// TwinCAT 3 PLC project Fraktal_Modules
// Title: Fraktal_Modules
// Company: fraktal-automation
// Author: fraktal-automation
// ProjectVersion: 0.11.0.3
// Description: Reusable Fraktal module library: cylinder CMs, clamp EM, simulation models, and configured device presets. Reason bands 10100s/11000s per Core 8.8.
// ProgramVersion: 3.1.4026.24
// libraries:
//   Fraktal_Core, 0.25.0.0 (fraktal-automation)
//   Tc2_MC2, * (Beckhoff Automation GmbH)
//   Tc2_Standard, * (Beckhoff Automation GmbH)
//   Tc2_System, * (Beckhoff Automation GmbH)
//   Tc2_Utilities, * (Beckhoff Automation GmbH)
//   Tc3_Module, * (Beckhoff Automation GmbH)
// project tree:
//   DUTs/ E_ConfigurableCylinderCommand.TcDUT (not stored), E_ClampCommand.TcDUT (not stored), E_CylinderCommand.TcDUT (not stored), E_CylinderPosition.TcDUT (not stored), E_PowerGroupCommand.TcDUT (not stored), ST_TwoHandHal.TcDUT (not stored), ST_TwoHandParCfg.TcDUT (not stored), ST_TwoHandParCmd.TcDUT (not stored), ST_TwoHandOutCmd.TcDUT (not stored), ST_TwoHandOutImm.TcDUT, ST_PowerGroupHal.TcDUT (not stored), ST_PowerGroupParCfg.TcDUT (not stored), ST_PowerGroupParCmd.TcDUT (not stored), ST_PowerGroupOutCmd.TcDUT (not stored), ST_PowerGroupOutImm.TcDUT, ST_ConfigurableCylinderParCfg.TcDUT (not stored), ST_ConfigurableCylinderParCmd.TcDUT (not stored), ST_ConfigurableCylinderOutCmd.TcDUT (not stored), ST_ConfigurableCylinderOutImm.TcDUT, ST_ConfigurableCylinderHal.TcDUT (not stored), ST_ClampParCfg.TcDUT (not stored), ST_ClampParCmd.TcDUT (not stored), ST_ClampOutCmd.TcDUT (not stored), ST_ClampOutImm.TcDUT, ST_CylinderHal.TcDUT (not stored), E_AxisCommand.TcDUT, ST_AxisParCfg.TcDUT, ST_AxisStationCfg.TcDUT, E_RobotOpMode.TcDUT, E_RobotJogMode.TcDUT, E_RobotCommand.TcDUT, E_RobotSimFault.TcDUT, ST_RobotParCfg.TcDUT, ST_RobotParCmd.TcDUT, ST_RobotOutCmd.TcDUT, ST_RobotOutImm.TcDUT, ST_StaubliConnParCfg.TcDUT, ST_RobotPose.TcDUT, E_HelpRole.TcDUT, E_MoveClass.TcDUT, ST_ApproachStep.TcDUT, ST_Corridor.TcDUT, ST_HelpAffinity.TcDUT, ST_NestHelpAffinity.TcDUT, ST_RouteGraph.TcDUT, ST_RobotGeometry.TcDUT, ST_RobotPoint.TcDUT, ST_RobotPointList.TcDUT, ST_AxisParCmd.TcDUT, ST_AxisOutCmd.TcDUT, ST_AxisOutImm.TcDUT, E_SeparatorCommand.TcDUT, E_SeparatorMode.TcDUT, ST_SeparatorHal.TcDUT, ST_SeparatorParCfg.TcDUT, ST_SeparatorParCmd.TcDUT, ST_SeparatorOutCmd.TcDUT, ST_SeparatorOutImm.TcDUT, ST_CylinderParCfg.TcDUT (not stored), ST_CylinderParCmd.TcDUT (not stored), ST_CylinderOutCmd.TcDUT (not stored), ST_CylinderOutImm.TcDUT, ST_CylinderIoIdentity.TcDUT (not stored), ST_DigitalInputHal.TcDUT (not stored), ST_DigitalInputParCfg.TcDUT, ST_DigitalInputParCmd.TcDUT, ST_DigitalInputOutCmd.TcDUT, ST_DigitalInputOutImm.TcDUT, ST_AirPressureHal.TcDUT (not stored), ST_AirPressureStationCfg.TcDUT, ST_AirPressureParCfg.TcDUT, ST_AirPressureParCmd.TcDUT, ST_AirPressureOutCmd.TcDUT, ST_AirPressureOutImm.TcDUT
//   Interfaces/ I_RobotConnector.TcIO
//   / FB_StaubliVal3Connector.TcPOU, FB_RobotRoutePlanner.TcPOU, FB_RobotCM.TcPOU, FB_SimRobotConnector.TcPOU, FB_AxisCM.TcPOU, FB_SeparatorCM.TcPOU, FB_ConfigurableCylinderCM.TcPOU, FB_ConfigurableCylinderSim.TcPOU, FB_ClampEM.TcPOU, FB_CylinderCM.TcPOU, FB_DigitalInputCM.TcPOU, FB_AirPressureMonitorCM.TcPOU, FB_CylinderSim.TcPOU, FB_Iv3VisionCM.TcPOU (not stored), FB_Matrix220CM.TcPOU (not stored), FB_PowerGroupCM.TcPOU, FB_TwoHandStartCM.TcPOU
//   Params/ PL_RobotPlanner.TcGVL, PL_ModuleReasons.TcGVL
// real-time tasks:
//   TASK PlcTask: cycle T#10ms, priority 20, ADS port 350

// ---- DUTs/ST_TwoHandOutImm.TcDUT
TYPE ST_TwoHandOutImm :
STRUCT
    LeftPressed     : BOOL;
    RightPressed    : BOOL;
    SafeActive      : BOOL;
    Armed           : BOOL;
    StartPulse      : BOOL;
    FieldbusHealthy : BOOL;
END_STRUCT
END_TYPE

// ---- DUTs/ST_PowerGroupOutImm.TcDUT
TYPE ST_PowerGroupOutImm :
STRUCT
    Status     : ST_PowerGroupStatus;
END_STRUCT
END_TYPE

// ---- DUTs/ST_ConfigurableCylinderOutImm.TcDUT
TYPE ST_ConfigurableCylinderOutImm :
STRUCT
    Position   : E_CylinderPosition;
    AtHome     : BOOL;
    AtWork     : BOOL;
END_STRUCT
END_TYPE

// ---- DUTs/ST_ClampOutImm.TcDUT
TYPE ST_ClampOutImm :
STRUCT
    Clamped    : BOOL;
    Unclamped  : BOOL;
END_STRUCT
END_TYPE

// ---- DUTs/E_AxisCommand.TcDUT
{attribute 'qualified_only'}
// Annex G motion CM. NONE is the unset value: dispatch rejects it (S5.6).
TYPE E_AxisCommand : (
    NONE    := 0,
    HOME    := 1,
    MOVE_TO := 2,
    // HELD commands (§7.6.1). Two entries rather than one plus a direction, so
    // the generic HMI renders two hold-buttons with no axis-specific code.
    // They never reach _M_Dispatch: a jog is not an Execute/Done command, and
    // PLCopen models it with level inputs for the same reason.
    JOG_POS := 3,
    JOG_NEG := 4
) DINT;
END_TYPE

// ---- DUTs/ST_AxisParCfg.TcDUT
// Core S3.8: SchemaVersion FIRST. Soft limits and dynamics are recipe/config,
// never sequence literals (S10.3) - scaling and hard limits stay in the axis
// configuration where the drive integrator owns them.
TYPE ST_AxisParCfg :
STRUCT
    SchemaVersion : UINT := 1;
    SoftMin       : LREAL := 0.0;
    SoftMax       : LREAL := 100.0;
    Velocity      : LREAL := 50.0;
    Acceleration  : LREAL := 500.0;
    Deceleration  : LREAL := 500.0;
    MoveTimeout   : TIME := T#10S;
    HomeTimeout   : TIME := T#30S;
    // Teach jog (§7.6.1). JogVelocity is DEFENCE IN DEPTH, not the protection:
    // the safety-rated reduced speed is the drive's own SLS or the cell's safe
    // speed monitor, because a scan overrun or a download must not be able to
    // remove the limit that keeps a person safe (§9).
    JogVelocity     : LREAL := 5.0;
    JogAcceleration : LREAL := 100.0;
    // How long a held request may go unheard before the axis stops. This is the
    // backstop for a stalled transport, NOT the normal stop: releasing the
    // control sends Dir=0 and stops immediately (O10).
    JogTimeout      : TIME := T#200MS;
END_STRUCT
END_TYPE

// ---- DUTs/ST_AxisStationCfg.TcDUT
// Core §3.8a/§3.8b - deployment data for one axis: what this MACHINE is, as
// opposed to what the current product needs. A taught position belongs here and
// not in ParCfg, because I_RecipeProvider loads and never stores: the next
// changeover would overwrite a number an operator spent time teaching.
//
// SchemaVersion is FIRST and is mandatory (§3.8b). Version 0 means never
// written - a first boot has lost nothing. Any OTHER unrecognized version means
// a real image was rejected, which is annunciated, because the difference
// between an empty machine and one that has just lost its commissioning is
// exactly what an operator needs told.
TYPE ST_AxisStationCfg :
STRUCT
    SchemaVersion  : UINT;      // 0 = never written; 2 = this layout
    TaughtPosition : LREAL;     // captured from the live ActPos (§3.8c)
    // v2. Does THIS INSTALLATION have a safety-rated enabling device for manual
    // motion? A deployment fact, not a preference, which is why it is station
    // configuration (§3.8a) rather than a recipe value or a compiled-in
    // assumption in the reusable type.
    //
    // TRUE - the default, and what every restore that predates this member and
    // every rejected image falls back to - keeps the §G.4a rule: no enabling
    // device permitting, no jog. FALSE says this installation has none, and a
    // station shall declare that only when it is true AND the consequence has
    // been assessed: a bench with a low-force motor on a desk is the case it
    // exists for, a cell with a person inside it is not. A station declaring
    // FALSE should declare a §7.5 engineering gate with it, so the machine
    // annunciates the departure instead of hiding it in a value nobody reads.
    JogRequiresEnable : BOOL;
END_STRUCT
END_TYPE

// ---- DUTs/E_RobotOpMode.TcDUT
// Annex I I.4a(a) - the robot CONTROLLER's operating mode, which bounds what
// motion is physically allowed. The PLC REQUESTS a mode and publishes separately
// what the controller REPORTS it actually is: a request that was not granted must
// stay visibly ungranted, never overwritten by optimism. UNKNOWN = 0 so an
// uninitialised value is never mistaken for a permissive mode.
{attribute 'qualified_only'}
TYPE E_RobotOpMode :
(
    UNKNOWN        := 0,
    AUTO_REMOTE    := 1,
    MANUAL_REDUCED := 2,
    MANUAL_HIGH    := 3
) DINT;
END_TYPE

// ---- DUTs/E_RobotJogMode.TcDUT
// Annex I I.3 - jog frame for manual motion. Named E_RobotJogMode, not
// E_JogMode: the short name collides with a Beckhoff motion-library type and the
// ambiguity surfaces only in a consumer that references both. Manual only, release-gated (S7.6).
{attribute 'qualified_only'}
TYPE E_RobotJogMode :
(
    JOINT     := 0,
    CARTESIAN := 1,
    TOOL      := 2
) DINT;
END_TYPE

// ---- DUTs/E_RobotCommand.TcDUT
// Annex I I.4 - the robot CM's command vocabulary. A point, a taught path, a
// generated route or a pallet nest is ONE command that runs to completion, so the
// robot looks identical to any other CM (S6.1). IDs are the only addressing.
{attribute 'qualified_only'}
TYPE E_RobotCommand :
(
    NONE           := 0,
    POWER_ON       := 1,
    POWER_OFF      := 2,
    HOME           := 3,
    MOVE_TO        := 4,   // one taught point, by ID
    RUN_PATH       := 5,   // a stored list, by ID and optional sub-range
    RUN_PALLET     := 6,   // one nest of a generated pallet grid
    MOVE_TEMPLATE  := 7,   // route generated by the help/nest graph (I.9)
    MOVE_FROM_AREA := 8,   // start resolved live from the current area (I.11)
    SET_TOOL       := 9,
    SET_FRAME      := 10,
    RECONNECT      := 11   // §3.15.4 deliberate reconnect; never resumes a command
) DINT;
END_TYPE

// ---- DUTs/E_RobotSimFault.TcDUT
// Annex I I.5c - the failures the simulation connector can be told to inject.
// Bounded and enumerated (O10): the reasons of I.2 are exactly what cannot be
// proven against a real arm without deliberately breaking a cell, so the sim
// must be able to produce them on demand - but only the ones some test or
// commissioning rehearsal actually needs, never a knob per reason.
{attribute 'qualified_only'}
TYPE E_RobotSimFault :
(
    NONE            := 0,
    POINT_UNREACHABLE := 1,   // the next motion command is refused before it starts
    NO_ROUTE          := 2,   // the next template move finds no path (I.9)
    LINK_LOSS         := 3,   // the heartbeat fails; the base drops and re-backs off
    PROTECTIVE_STOP   := 4,   // the crash device trips, in motion or at rest
    NOT_RESUMABLE     := 5    // a held move cannot resume - the arm left the path (I.4b)
) DINT;
END_TYPE

// ---- DUTs/ST_RobotParCfg.TcDUT
// Recipe-class configuration (S3.8), versioned.
TYPE ST_RobotParCfg :
STRUCT
    SchemaVersion : UINT := 1;
    MoveTimeout   : TIME := T#60S;   // per-command guard; the Unit step's ExpectedTime (S6.5) remains the outer one
    HomeTimeout   : TIME := T#120S;
    SpeedScaleMin : REAL := 1.0;     // band a recipe SpeedScale is validated against (I.4a(b))
    SpeedScaleMax : REAL := 100.0;
    // Ceiling per controller operating mode; the CM applies MIN(ceiling, ParCmd.SpeedScale).
    // UNKNOWN = 0 so an unreported mode yields the safest ceiling, not the fastest.
    // Indexed by E_RobotOpMode's ordinals - UNKNOWN, AUTO_REMOTE,
    // MANUAL_REDUCED, MANUAL_HIGH. UNKNOWN is 0.0 on purpose: a mode the
    // controller has not reported never earns a speed allowance.
    SpeedCeiling  : ARRAY[0..3] OF REAL := [0.0, 100.0, 25.0, 100.0];
END_STRUCT
END_TYPE

// ---- DUTs/ST_RobotParCmd.TcDUT
// Latched by the base on the Execute rising edge (S6.1). No Offset field yet:
// the runtime-correction exception of I.8a is deferred with the connector support
// for it - declaring a field no consumer reads would be dead surface, and an
// unvalidated offset would be worse (S14).
TYPE ST_RobotParCmd :
STRUCT
    TargetId   : DWORD := 0;   // point / list / pallet / tool / frame - or the TO position
    FromId     : DWORD := 0;   // FROM position (MOVE_TEMPLATE only)
    Nest       : DINT := 0;    // nest index (RUN_PALLET only)
    StartIdx   : DINT := -1;   // sub-path bounds (RUN_PATH; -1,-1 = whole list)
    EndIdx     : DINT := -1;
    SpeedScale : REAL := 100.0;   // process speed for THIS command, % of taught (I.4a(b))
    AcknowledgeController : BOOL; // RECONNECT also clears the robot's own fault
END_STRUCT
END_TYPE

// ---- DUTs/ST_RobotOutCmd.TcDUT
// Valid on Done (S3.10).
TYPE ST_RobotOutCmd :
STRUCT
    ReachedId : DWORD;   // position actually reached
END_STRUCT
END_TYPE

// ---- DUTs/ST_RobotOutImm.TcDUT
// Cyclic live status mirrored from the connector, plus the first-out diagnostic.
TYPE ST_RobotOutImm :
STRUCT
    Linked         : BOOL;
    Referenced     : BOOL;
    MotionBusy     : BOOL;           // the ARM is moving - not the command handshake
    ActualMode     : E_RobotOpMode;  // what the controller REPORTS (I.4a(a))
    CurrentArea    : DWORD;          // 0 = none/undefined (I.11)
    ProtectiveStop : BOOL;           // process protection, NOT S9 safety (I.4a(c))
    Resumable      : BOOL;           // resume still valid on the retained path (I.4b)
    SpeedScale     : REAL;           // scale actually in force
END_STRUCT
END_TYPE

// ---- DUTs/ST_StaubliConnParCfg.TcDUT
// Deployment configuration for the VAL3 connector (S3.8a station config).
TYPE ST_StaubliConnParCfg :
STRUCT
    SchemaVersion : UINT := 1;
    Host          : STRING(80);
    Port          : UINT := 11000;      // VAL3 fraktal_server command socket
    Terminator    : STRING(2) := '$R';  // ASCII 13, as the Staubli sioLink default
    RespTimeout   : TIME := T#2S;       // per-request; motion completion is polled, not awaited
    StatusPeriod  : TIME := T#100MS;    // idle status poll interval
END_STRUCT
END_TYPE

// ---- DUTs/ST_RobotPose.TcDUT
// Annex I I.3 - one pose type for live readback, taught geometry and runtime
// corrections. The connector owns the Euler convention and the units it speaks
// to the controller in; per-model facts like that are data it reads, never
// branches in application code.
TYPE ST_RobotPose :
STRUCT
    X  : LREAL;   // mm
    Y  : LREAL;
    Z  : LREAL;
    RX : LREAL;   // deg
    RY : LREAL;
    RZ : LREAL;
END_STRUCT
END_TYPE

// ---- DUTs/E_HelpRole.TcDUT
// Annex I I.10 - which direction of travel a help corridor is legal for.
// EITHER is 0 so a zero-initialized corridor is bidirectional: a nest is
// exit-able the way it was entered unless its geometry is physically one-way.
{attribute 'qualified_only'}
TYPE E_HelpRole :
(
    EITHER   := 0,
    APPROACH := 1,
    DEPART   := 2
) DINT;
END_TYPE

// ---- DUTs/E_MoveClass.TcDUT
// Annex I I.10.2 - how a generated step is flown. The class selects the motion
// mode AND which configured velocity applies, so speed stays configuration
// (I.4a(b)) and never becomes a literal in the route graph.
{attribute 'qualified_only'}
TYPE E_MoveClass :
(
    SLOW_LINEAR := 0,
    FAST_PTP    := 1,
    SLOW_JOINTS := 2
) DINT;
END_TYPE

// ---- DUTs/ST_ApproachStep.TcDUT
// Annex I I.10.2 - one offset from the nest pose, in the nest's own frame.
TYPE ST_ApproachStep :
STRUCT
    D         : ST_RobotPose;   // offset applied to the nest pose
    MoveClass : E_MoveClass;
END_STRUCT
END_TYPE

// ---- DUTs/ST_Corridor.TcDUT
// Annex I I.10.2 - how a nest is entered from, or left toward, one serving
// help. Steps are stored nest-ward -> help-ward: a DEPART corridor emits them
// in that order, an APPROACH corridor emits them reversed and then the nest.
// StepCount = 0 with ListId <> 0 names a taught list instead, for geometry a
// few axis offsets cannot express.
TYPE ST_Corridor :
STRUCT
    Steps     : ARRAY[1..PL_RobotPlanner.MAX_APPROACH_STEPS] OF ST_ApproachStep;
    StepCount : INT;
    ListId    : DWORD;
END_STRUCT
END_TYPE

// ---- DUTs/ST_HelpAffinity.TcDUT
// Annex I I.10 - one help point serving a nest, with the direction it is legal
// for and the transit region it connects to. Region is needed only where a nest
// has two corridors for the SAME direction; most nests need only the role.
TYPE ST_HelpAffinity :
STRUCT
    HelpId   : INT;          // index into the help arrays; 0 = unused entry
    Role     : E_HelpRole;
    RegionId : DWORD;        // 0 = any
    Approach : ST_Corridor;  // how the nest is ENTERED from this help
    Depart   : ST_Corridor;  // how it is LEFT toward this help - not the approach reversed
END_STRUCT
END_TYPE

// ---- DUTs/ST_NestHelpAffinity.TcDUT
// Annex I I.10 - the help points serving one nest. Count = 1 is the trivial
// single-help case; multi-help is the general one.
TYPE ST_NestHelpAffinity :
STRUCT
    Helps : ARRAY[1..PL_RobotPlanner.MAX_HELPS_PER_NEST] OF ST_HelpAffinity;
    Count : INT;
END_STRUCT
END_TYPE

// ---- DUTs/ST_RouteGraph.TcDUT
// Annex I I.9 / Core S10.7 - the declarative routing model. The application
// supplies configuration, not traversal code: one generic planner resolves it
// for every station.
TYPE ST_RouteGraph :
STRUCT
    // help <-> help adjacency: which transits are allowed
    HelpAdj    : ARRAY[1..PL_RobotPlanner.MAX_HELPS, 1..PL_RobotPlanner.MAX_HELPS] OF BOOL;
    // the transit region each help belongs to; used only to break ties between
    // same-direction corridors (I.10)
    HelpRegion : ARRAY[1..PL_RobotPlanner.MAX_HELPS] OF DWORD;
    // per gripper, per nest: one OR MORE serving help points (I.10, I.12)
    NestHelp   : ARRAY[1..PL_RobotPlanner.MAX_GRIPPERS, 1..PL_RobotPlanner.MAX_NESTS] OF ST_NestHelpAffinity;
    // optional taught nest -> nest list, bypassing the help routing entirely
    DirectNest : ARRAY[1..PL_RobotPlanner.MAX_NESTS, 1..PL_RobotPlanner.MAX_NESTS] OF DWORD;
END_STRUCT
END_TYPE

// ---- DUTs/ST_RobotGeometry.TcDUT
// Annex I I.1 - taught geometry held as Fraktal configuration and pushed to the
// controller by the connector, so it lives inside changeover (S3.8), parameter
// sets (S3.8b), access control (S7.7) and audit (S8.3) rather than only inside a
// vendor engineering tool. Editable through bounded collection capabilities
// (S3.10.2a) with pose cells filled by teach capture (S3.8c).
TYPE ST_RobotGeometry :
STRUCT
    HelpPose : ARRAY[1..PL_RobotPlanner.MAX_HELPS] OF ST_RobotPose;
    NestPose : ARRAY[1..PL_RobotPlanner.MAX_GRIPPERS, 1..PL_RobotPlanner.MAX_NESTS] OF ST_RobotPose;
END_STRUCT
END_TYPE

// ---- DUTs/ST_RobotPoint.TcDUT
// Annex I I.8 - one element of a generated or taught route. A point either
// names a pose to move to, or (ListId <> 0) a taught list for the executor to
// run at that place in the sequence.
TYPE ST_RobotPoint :
STRUCT
    Target    : ST_RobotPose;
    MoveClass : E_MoveClass;
    ListId    : DWORD;    // 0 = move to Target; otherwise run this taught list
END_STRUCT
END_TYPE

// ---- DUTs/ST_RobotPointList.TcDUT
// Annex I I.8 - a bounded generated or taught route.
TYPE ST_RobotPointList :
STRUCT
    Points : ARRAY[1..PL_RobotPlanner.MAX_ROUTE_POINTS] OF ST_RobotPoint;
    Count  : INT;
END_STRUCT
END_TYPE

// ---- DUTs/ST_AxisParCmd.TcDUT
// Latched by the base on the Execute rising edge (S6.1).
TYPE ST_AxisParCmd :
STRUCT
    Target : LREAL;   // absolute target for MOVE_TO, in axis units
END_STRUCT
END_TYPE

// ---- DUTs/ST_AxisOutCmd.TcDUT
// Valid on Done (S3.12).
TYPE ST_AxisOutCmd :
STRUCT
    InPosition : BOOL;
    Homed      : BOOL;
END_STRUCT
END_TYPE

// ---- DUTs/ST_AxisOutImm.TcDUT
// Cyclic live status plus the first-out diagnostic (S3.12, S6.9).
TYPE ST_AxisOutImm :
STRUCT
    ActPos       : LREAL;
    ActVelocity  : LREAL;
    Homed        : BOOL;
    DriveEnabled : BOOL;
    // The stored taught position (S3.8b PERSISTENT), published beside the live
    // ActPos so an operator can compare what is stored with where the axis is
    // before capturing over it (S3.8c(b)).
    TaughtPosition : LREAL;
    Jogging      : BOOL;   // a held jog is driving the axis right now (§7.6.1)
    // Why the last jog stopped: 0 = released normally, otherwise the §8.8 reason.
    // Published status, deliberately NOT an alarm - a jog that stops because the
    // operator let go is the designed behaviour, and filing it as a fault would
    // fill the record with events that were never faults (§6.1).
    JogStopReason : DINT;
END_STRUCT
END_TYPE

// ---- DUTs/E_SeparatorCommand.TcDUT
{attribute 'qualified_only'}
// Annex A separator/stopper. NONE is the unset value: dispatch rejects it (S5.6).
TYPE E_SeparatorCommand : (
    NONE       := 0,
    SEPARATE   := 1,    // release exactly one carrier
    OPEN_CLOSE := 2     // hold the stopper open or closed per ParCmd.OpenStopper
) DINT;
END_TYPE

// ---- DUTs/E_SeparatorMode.TcDUT
{attribute 'qualified_only'}
// Separation behaviour variants (Annex A). SEPARATOR checks the carrier at AND
// after the device; STOPPER checks only at it.
TYPE E_SeparatorMode : (
    SEPARATOR  := 0,
    STOPPER    := 1,
    ASISTOPPER := 2,
    LEADFRAME  := 3
) DINT;
END_TYPE

// ---- DUTs/ST_SeparatorHal.TcDUT
// HAL view (S10.3). The driver owns invert/debounce and the raw %I/%Q symbols;
// the module only ever touches these clean signals, so simulation and hardware
// are the same code (S2.6).
TYPE ST_SeparatorHal :
STRUCT
    CarrierAt    : BOOL;   // input  - carrier present at the separator
    CarrierAfter : BOOL;   // input  - carrier present just past the separator
    OpenedFb     : BOOL;   // input  - separator-opened feedback (optional)
    ValveOpen    : BOOL;   // output - drives the open solenoid
END_STRUCT
END_TYPE

// ---- DUTs/ST_SeparatorParCfg.TcDUT
// Core S3.8: SchemaVersion FIRST, initialized to the expected version.
TYPE ST_SeparatorParCfg :
STRUCT
    SchemaVersion : UINT := 1;
    Mode          : E_SeparatorMode := E_SeparatorMode.SEPARATOR;
    CheckAfter    : BOOL := TRUE;    // require the carrier-after arrival/clear checks
    UsesOpenFb    : BOOL := FALSE;   // require the open feedback on OPEN_CLOSE
    MaxOpenTime   : TIME := T#3S;    // CarrierAt must clear within this after opening
    SOnMaxTime    : TIME := T#3S;    // CarrierAfter must arrive/clear within this
    CloseDelay    : TIME := T#0S;
    Timeout       : TIME := T#10S;   // overall command timeout
END_STRUCT
END_TYPE

// ---- DUTs/ST_SeparatorParCmd.TcDUT
// Latched by the base on the Execute rising edge (S6.1).
TYPE ST_SeparatorParCmd :
STRUCT
    OpenStopper : BOOL;   // OPEN_CLOSE: TRUE = open, FALSE = close
END_STRUCT
END_TYPE

// ---- DUTs/ST_SeparatorOutCmd.TcDUT
// Valid on Done (S3.12).
TYPE ST_SeparatorOutCmd :
STRUCT
    SeparateOk    : BOOL;
    SeparatorOpen : BOOL;
END_STRUCT
END_TYPE

// ---- DUTs/ST_SeparatorOutImm.TcDUT
// Cyclic live status plus the first-out diagnostic (S3.12, S6.9).
TYPE ST_SeparatorOutImm :
STRUCT
    CarrierAt    : BOOL;
    CarrierAfter : BOOL;
    OpenedFb     : BOOL;
    ValveOpen    : BOOL;
END_STRUCT
END_TYPE

// ---- DUTs/ST_CylinderOutImm.TcDUT
TYPE ST_CylinderOutImm :
STRUCT
    Extended   : BOOL;
    Retracted  : BOOL;
    ExtendedSensorTag : STRING(80);
    RetractedSensorTag: STRING(80);
    ExtendOutputTag   : STRING(80);
    RetractOutputTag  : STRING(80);
END_STRUCT
END_TYPE

// ---- DUTs/ST_DigitalInputParCfg.TcDUT
TYPE ST_DigitalInputParCfg :
STRUCT
    SchemaVersion : UINT := 1; // §3.8: first member even when the passive type has no behavior parameter
END_STRUCT
END_TYPE

// ---- DUTs/ST_DigitalInputParCmd.TcDUT
TYPE ST_DigitalInputParCmd :
STRUCT
    Reserved : BOOL; // passive monitor: physical four-structure contract, no command payload
END_STRUCT
END_TYPE

// ---- DUTs/ST_DigitalInputOutCmd.TcDUT
TYPE ST_DigitalInputOutCmd :
STRUCT
    Reserved : BOOL; // passive monitor: no command result
END_STRUCT
END_TYPE

// ---- DUTs/ST_DigitalInputOutImm.TcDUT
TYPE ST_DigitalInputOutImm :
STRUCT
    Value : BOOL;
    Quality : BOOL;
    IoTag : STRING(80);
END_STRUCT
END_TYPE

// ---- DUTs/ST_AirPressureStationCfg.TcDUT
// Core §3.8a/§3.8b — deployment data for this monitor. The qualification time
// depends on the physical switches and the air system they sit in, not on the
// product being made, so it is station configuration and NOT part of any model
// recipe: it must not change at changeover, and it must survive a restart.
// SchemaVersion stays first (§3.8b) so a retained image from another layout is
// rejected and re-initialized instead of read by field position.
TYPE ST_AirPressureStationCfg :
STRUCT
    SchemaVersion : UINT := 1;
    ConflictTime  : TIME := T#500MS; // qualify contradictory mechanical switches
END_STRUCT
END_TYPE

// ---- DUTs/ST_AirPressureParCfg.TcDUT
// v2 moved ConflictTime to ST_AirPressureStationCfg: it varies per
// deployment, not per model, and §3.8a places such a value in station
// configuration. This monitor has no model data of its own, so what remains
// is the versioned shell the §3.12 contract asks every module to carry.
TYPE ST_AirPressureParCfg :
STRUCT
    SchemaVersion : UINT := 2;       // §3.8: MUST remain first
END_STRUCT
END_TYPE

// ---- DUTs/ST_AirPressureParCmd.TcDUT
TYPE ST_AirPressureParCmd :
STRUCT
    Reserved : BOOL; // passive monitor: physical four-structure contract, no command payload
END_STRUCT
END_TYPE

// ---- DUTs/ST_AirPressureOutCmd.TcDUT
TYPE ST_AirPressureOutCmd :
STRUCT
    Reserved : BOOL; // passive monitor: no command result
END_STRUCT
END_TYPE

// ---- DUTs/ST_AirPressureOutImm.TcDUT
TYPE ST_AirPressureOutImm :
STRUCT
    LowPressure : BOOL;
    OperatingPressure : BOOL;
    PressureOk : BOOL;
    Contradictory : BOOL;
    Quality : BOOL;
    LowSensorTag : STRING(80);
    OperatingSensorTag : STRING(80);
END_STRUCT
END_TYPE

// ---- Params/PL_RobotPlanner.TcGVL
{attribute 'qualified_only'}
// Annex I - bounds for the declarative routing model. Every structure the
// planner touches is statically sized (Core S1.1 O10): a route that would
// exceed MAX_ROUTE_POINTS is refused, never allocated.
VAR_GLOBAL CONSTANT
    MAX_HELPS           : INT := 8;    // transit / wait positions
    MAX_NESTS           : INT := 16;   // work positions, per gripper
    MAX_GRIPPERS        : INT := 4;    // nests are per-gripper (I.12); 1 is the trivial case
    MAX_HELPS_PER_NEST  : INT := 4;    // serving corridors on one nest (I.10)
    MAX_APPROACH_STEPS  : INT := 4;    // offset steps in one corridor (I.10.2)
    MAX_ROUTE_POINTS    : INT := 32;   // generated route length
END_VAR

// ---- Params/PL_ModuleReasons.TcGVL
{attribute 'qualified_only'}
// Core §8.8 band constants (band-extensibility rule): cylinder CM 10100-10199,
// clamp EM 11000-11999 — registered in the Core §8.8 registry.
VAR_GLOBAL CONSTANT
    CYL_NOT_EXTENDED    : DINT := 10101;
    CYL_NOT_RETRACTED   : DINT := 10102;
    CYL_BOTH_SENSORS    : DINT := 10103;
    CLAMP_NOT_CONFIRMED : DINT := 11001;
    // basic cylinder 10110-10119
    CYL_HOME_NOT_REACHED : DINT := 10111;   // timeout moving to home
    CYL_WORK_NOT_REACHED : DINT := 10112;   // timeout moving to work
    CYL_POS_IMPLAUSIBLE  : DINT := 10113;   // home AND work sensor confirmed at once (implausible)
    CYL_SENSOR_LOST      : DINT := 10114;   // confirmed position sensor dropped while holding
    CYL_DISCREPANCY      : DINT := 10116;   // redundant sensors for one position disagree > DiscrepancyTime
    CYL_CFG_INVALID      : DINT := 10115;   // TravelTime >= MoveTimeout, or no sensor+no travel
    // axis CM 10201-10206 (Annex G)
    AXIS_TARGET_OOR      : DINT := 10201;   // target outside soft limits (rejected)
    AXIS_MOVE_TIMEOUT    : DINT := 10202;   // MC move did not complete within the timeout
    AXIS_DRIVE_FAULT     : DINT := 10203;   // MC_* .Error / drive fault
    AXIS_NOT_HOMED       : DINT := 10204;   // MOVE_TO before a valid home
    AXIS_JOG_NOT_ENABLED : DINT := 10205;   // teach jog asked with no enabling device held
    AXIS_JOG_RELEASED    : DINT := 10206;   // the held jog request stopped arriving
    // power-group CM 10500-10599
    POWER_ENABLE_WITHHELD : DINT := 10501;
    POWER_FEEDBACK_TIMEOUT: DINT := 10502;
    // separator/stopper CM 10001-10005 (Annex A)
    SEP_NO_CARRIER_AT       : DINT := 10001;   // carrier never present at the separator
    SEP_CARRIER_NOT_CLEARED : DINT := 10002;   // CarrierAt did not clear after opening
    SEP_CARRIER_NOT_ARRIVED : DINT := 10003;   // CarrierAfter did not arrive in time
    SEP_NOT_OPENED_FB       : DINT := 10004;   // open feedback missing
    SEP_SON_NOT_CLEARED     : DINT := 10005;   // CarrierAfter did not clear after close
    // robot route planner 10301-10315 (Annex I) - only what the planner raises today
    ROBOT_POINT_UNREACHABLE  : DINT := 10301;   // taught point not reachable with the active tool/frame
    ROBOT_MOVE_TIMEOUT       : DINT := 10303;   // motion did not complete within ParCfg timeout
    ROBOT_CONTROLLER_FAULT   : DINT := 10304;   // drive/controller fault reported by the robot itself
    ROBOT_NOT_REFERENCED     : DINT := 10305;   // motion commanded before a valid home/reference
    ROBOT_NO_ROUTE           : DINT := 10308;   // help graph defines no path between the two positions
    ROBOT_NO_HELP_FOR_NEST   : DINT := 10310;   // no help point resolves for a nest given the move endpoints
    ROBOT_MODE_NOT_PERMITTED : DINT := 10311;   // controller mode does not permit this command
    ROBOT_PROTECTIVE_STOP    : DINT := 10313;   // collision/crash device tripped - NOT a S9 safety function
    ROBOT_PARAM_OOR          : DINT := 10314;   // a command parameter is outside its configured band
    ROBOT_RESUME_INVALID     : DINT := 10315;   // resume after hold, but the arm left the retained path
    // air-pressure monitor CM 10600-10699
    AIR_SWITCH_CONFLICT    : DINT := 10601;
END_VAR

// ---- Interfaces/I_RobotConnector.TcIO
// Annex I I.3 - the primitive robot surface, below the robot CM and above the
// protocol. Everything under it (transport, point database, kinematics, path
// planning) is confined to the implementation (Core S3.15).
//
// MOST OF THIS SURFACE IS NOT FRAKTAL'S TO DEFINE. SRCI (Standard Robot Command
// Interface, PROFIBUS/PROFINET International) already standardises the PLC/robot
// command boundary, so the members below are DEFINED BY their SRCI equivalent and
// are not re-described here - re-describing them would create a second authority
// for someone else's contract and guarantee drift (S1.1 O9). The mapping is
// normative and lives in Annex I I.3:
//
//   PowerOn/PowerOff  = EnableRobot        Interrupt/Resume = GroupInterrupt/Continue
//   Home              = referencing        Abort            = GroupStop
//   MoveToPoint       = MoveDirectAbsolute ResetController  = GroupReset
//   RunPath           = sequential moves   RequestMode      = SetOperationMode
//   ActualPosition    = ReadActualPosition SetSpeedScale    = ChangeSpeedOverride
//   ControllerMessage = ReadMessages       SetTool/SetFrame = Read Tool/FrameData
//   SetPayload        = Read/WriteLoadData Jog              = GroupJog
//
// Seven members have NO SRCI equivalent, because they express this annex's own
// model: RunPallet, MoveTemplate, MoveFromArea, CurrentArea, ProtectiveStop,
// Resumable and LastResult. They are what the standard adds over an ordinary
// robot command interface.
//
// Every method returns immediately: FALSE means the request was refused outright
// (unknown id, unreachable, no route, not linked) and LastResult carries the
// first-out reason. Motion progress is observed over scans via Busy, never awaited.
INTERFACE I_RobotConnector EXTENDS I_DeviceConnector

// SRCI EnableRobot (Core). Arm power on.
METHOD PowerOn : BOOL
END_METHOD

// SRCI EnableRobot (Core). Arm power off.
METHOD PowerOff : BOOL
END_METHOD

// SRCI referencing. Drive to the home/reference configuration.
METHOD Home : BOOL
END_METHOD

// SRCI MoveDirectAbsolute/MoveLinearAbsolute, target resolved from the ID.
METHOD MoveToPoint : BOOL
VAR_INPUT
    PointId : DWORD;
END_VAR
END_METHOD

// Sequential SRCI moves over a stored list. (-1,-1) = the whole list.
METHOD RunPath : BOOL
VAR_INPUT
    ListId   : DWORD;
    StartIdx : DINT;
    EndIdx   : DINT;
END_VAR
END_METHOD

// SRCI GroupInterrupt (Core). Stop ON PATH, retaining the resume point - the
// robot half of the S6.1 HELD contract (I.4b). A cylinder honours HELD by
// de-energising; a robot cannot, because resuming a 26-point path by
// re-commanding it would re-run executed points or approach from an untaught pose.
METHOD Interrupt : BOOL
END_METHOD

// SRCI GroupContinue (Core). Continue FROM the retained path point. Callers
// must check Resumable first: resuming onto a path the tool has left is how a
// robot drives through a fixture (I.4b).
METHOD Resume : BOOL
END_METHOD

// SRCI GroupStop (Core). Commands are NOT auto-repeated; resumption is
// deliberate (Annex D / S9.3).
METHOD Abort : BOOL
END_METHOD

// SRCI GroupReset (Core). Acknowledge the robot's OWN messages. Without this a
// controller fault can be detected but never cleared.
METHOD ResetController : BOOL
END_METHOD

// SRCI SetOperationMode (Core). REQUEST only - the controller grants. Compare
// with ActualMode, which reports what it actually is (I.4a(a)).
METHOD RequestMode : BOOL
VAR_INPUT
    Mode : E_RobotOpMode;
END_VAR
END_METHOD

// SRCI ChangeSpeedOverride (Core). Ceiling on path speed, as a percentage of
// taught. The CM applies MIN(mode ceiling, recipe scale) (I.4a(b)).
METHOD SetSpeedScale : BOOL
VAR_INPUT
    Percent : REAL;
END_VAR
END_METHOD

// SRCI ReadToolData (Core) - selection by ID. Geometry stays taught data.
METHOD SetTool : BOOL
VAR_INPUT
    ToolId : DWORD;
END_VAR
END_METHOD

// SRCI ReadFrameData (Core) - selection by ID. The frame may be chained (I.12).
METHOD SetFrame : BOOL
VAR_INPUT
    FrameId : DWORD;
END_VAR
END_METHOD

// SRCI Read/WriteLoadData. The active load case, which changes the moment a part
// is gripped or released; a move computed for the wrong mass degrades accuracy
// and brake margin silently (I.3).
METHOD SetPayload : BOOL
VAR_INPUT
    LoadId : DWORD;
END_VAR
END_METHOD

// SRCI GroupJog (Core). Manual only, release-gated (S7.6), and refused unless
// ActualMode is a manual mode (I.4a(a)).
METHOD Jog : BOOL
VAR_INPUT
    Mode : E_RobotJogMode;
    Axis : INT;
    Dir  : INT;
END_VAR
END_METHOD

// NO SRCI EQUIVALENT. One nest of a generated pallet grid, addressed by pallet
// ID and nest index; the grid itself is generated from taught corners (I.12).
METHOD RunPallet : BOOL
VAR_INPUT
    PalletId : DWORD;
    Nest     : DINT;
END_VAR
END_METHOD

// NO SRCI EQUIVALENT. Route generated by the declarative help/nest graph between
// two KNOWN positions (I.9) - the PLC names from and to, never the waypoints.
METHOD MoveTemplate : BOOL
VAR_INPUT
    FromPosId : DWORD;
    ToPosId   : DWORD;
END_VAR
END_METHOD

// NO SRCI EQUIVALENT. Route planned from WHICHEVER planning area the TCP
// currently occupies, resolved live. The application's primary motion command,
// because it needs no assumption about the start pose; pose recovery after an
// E-stop is its extreme case, not a separate mode (I.11).
METHOD MoveFromArea : BOOL
VAR_INPUT
    ToPosId : DWORD;
END_VAR
END_METHOD

// The ROBOT is executing motion. Deliberately NOT called Busy: the module base
// already publishes Busy for its own command handshake, and the two are different
// questions - "is my command running" versus "is the arm moving".
PROPERTY MotionBusy : BOOL
GET
END_GET
END_PROPERTY

// A valid home/reference exists. MOVE/RUN before this is refused (S5.6).
PROPERTY Referenced : BOOL
GET
END_GET
END_PROPERTY

// What the controller REPORTS its operating mode to be - read-only status, and
// never treated as a safety grant (S9). Deliberately separate from the request.
PROPERTY ActualMode : E_RobotOpMode
GET
END_GET
END_PROPERTY

// SRCI ReadActualPosition (Core). Live TCP pose, for display and diagnostics.
// Reading a pose is not commanding one, so I.1's boundary is untouched.
PROPERTY ActualPosition : ST_RobotPose
GET
END_GET
END_PROPERTY

// SRCI ReadMessages (Core). The robot's OWN message, carried verbatim - what a
// service technician actually needs, rather than a Fraktal paraphrase.
PROPERTY ControllerMessage : ST_Diagnostic
GET
END_GET
END_PROPERTY

// NO SRCI EQUIVALENT. The planning area the TCP is in; 0 = none/undefined, which
// is what makes ROBOT_AREA_UNRESOLVED an explicit first-out instead of a silent
// stall (I.11).
PROPERTY CurrentArea : DWORD
GET
END_GET
END_PROPERTY

// NO SRCI EQUIVALENT. Collision/crash-protection device tripped. This is PROCESS
// protection, detected and acted on by the ordinary PLC - NOT a S9 safety
// function, and deliberately carrying its own reason so the alarm record does not
// misreport a process event as a safety event (I.4a(c)).
PROPERTY ProtectiveStop : BOOL
GET
END_GET
END_PROPERTY

// NO SRCI EQUIVALENT. Whether Resume is still valid on the retained path. A hold
// is exactly the window in which an operator is most likely to jog the arm - that
// is what the pause was for - so this turns "the arm was moved while suspended"
// into a clean refusal instead of a move through untaught space (I.4b).
PROPERTY Resumable : BOOL
GET
END_GET
END_PROPERTY

// First-out reason and SourcePath of the last refused or failed request, adopted
// verbatim by the owning CM's rollup (S8.2).
PROPERTY LastResult : ST_Diagnostic
GET
END_GET
END_PROPERTY

END_INTERFACE

// ---- FB_StaubliVal3Connector.TcPOU
// Annex I I.3/I.5 - Staubli VAL3 connector: one conformant implementation of
// I_RobotConnector, speaking a line protocol to a `fraktal_server` VAL3
// application on the robot controller.
//
// WHY TCP AND NOT uniVAL/EtherCAT. Both are conformant behind this interface and
// the parent Unit is unchanged either way (I.5), but only this one can be
// developed and regression-tested with NO ARM: the Staubli Robotics Suite
// Emulator answers the same TCP sockets as a real CS9 controller, whereas a
// virtual controller cannot present an EtherCAT slave. uniVAL plc over EtherCAT
// (Beckhoff TF5130) remains the production binding where cycle determinism
// matters; this one is what makes O6 - commissioning before hardware - true for
// a robot cell, and what S5.7 tests run against.
//
// A CONNECTOR, like FB_SimRobotConnector (Core §3.15.1): it is serviced by the
// robot CM it is composed in (§3.15.3), so swapping the two changes a declaration
// and not the module tree (I.5). Everything connector-shaped is INHERITED from
// FB_DeviceConnectorBase - session, heartbeat, loss confirmation after
// LinkTimeout, bounded reconnect with no self-resume (§3.15.2) - and the ASCII
// framing and one-outstanding-request rule are FB_AsciiLink's, shared with the
// device CMs (§1.1 O9). This type adds only the robot protocol.
//
// PROTOCOL (ASCII, one line per message, terminator from ParCfg):
//   request   <CMD>[,<arg>]...
//   response  <CMD>,OK[,<payload>]...   accepted / completed
//             <CMD>,ERR,<code>,<text>   refused or faulted by the controller
// Commands are ID-ADDRESSED (I.1): a point, list, pallet, tool, frame or load is
// named by its identifier and never by a coordinate. The single exception the
// standard permits - a bounded offset correction for a runtime-located target
// (I.8a) - is not implemented here yet and is not smuggled in.
//
// STATUS IS THE HEARTBEAT: every ParCfg.StatusPeriod the connector issues STA, so
// MotionBusy/Referenced/ActualMode/CurrentArea/ProtectiveStop/Resumable/pose stay
// current without the robot originating traffic, and a controller that stops
// answering is declared lost after LinkTimeout rather than trusted forever.
FUNCTION_BLOCK FB_StaubliVal3Connector EXTENDS FB_DeviceConnectorBase IMPLEMENTS I_RobotConnector
VAR_INPUT
    ParCfg : ST_StaubliConnParCfg;
END_VAR
VAR_OUTPUT
    LinkState    : E_ByteChannelState;   // the transport, for diagnosis
    LastResponse : STRING(255);          // the controller's last reply, verbatim
END_VAR
VAR
    {attribute 'OPC.UA.DA' := '0'}
    _link        : FB_AsciiLink;
    _busy        : BOOL;
    _referenced  : BOOL;
    _mode        : E_RobotOpMode;
    _reqMode     : E_RobotOpMode;
    _area        : DWORD;
    _protStop    : BOOL;
    _resumable   : BOOL;
    _pose        : ST_RobotPose;
    _ctrlMsg     : ST_Diagnostic;
    _lastResult  : ST_Diagnostic;
    _statusPend  : BOOL;   // the outstanding request is the heartbeat's STA
    _hbReply     : BOOL;   // a well-formed reply arrived since the heartbeat asked
END_VAR

Cyclic();

// Wire identity and transport. Called once from the composition root (S3.11);
// the robot CM then services the connector every scan (§3.15.3).
METHOD SetupLink : BOOL
VAR_INPUT
    Name    : STRING(80);
    Chan    : I_ByteChannel;
    DevHost : STRING(80);
    DevPort : UINT;
END_VAR
SetupLink := FALSE;
Setup(Name := Name);
IF (Chan = 0) OR (DevHost = '') THEN
    _lastResult.ReasonCode  := PL_TcpDevReasons.DEV_CFG_INVALID;
    _lastResult.Description := 'std.error.deviceConnectionNotConfigured';
    _lastResult.SourcePath  := Name;
    RETURN;
END_IF
ParCfg.Host := DevHost;
ParCfg.Port := DevPort;
SetupLink := _link.M_Bind(Chan := Chan);
END_METHOD

// Run the link and parse what it delivered, then let the base run the session,
// the heartbeat and the bounded reconnect exactly as for any connector.
METHOD Cyclic : BOOL
VAR
    evt : E_AsciiLinkEvent;
END_VAR
_link.Terminator := ParCfg.Terminator;
_link.RespTimeout := ParCfg.RespTimeout;
HbPeriod := ParCfg.StatusPeriod;
evt := _link.M_Tick();
LinkState := _link.State;
CASE evt OF
    E_AsciiLinkEvent.NONE:
        ;
    E_AsciiLinkEvent.RESPONSE:
        LastResponse := _link.LastResponse;
        _M_OnResponse(Response := _link.Response);
    E_AsciiLinkEvent.TIMEOUT:
        IF _statusPend THEN
            // An unanswered heartbeat is not a fault by itself: it stays PENDING,
            // and the base declares the link lost only after LinkTimeout (§3.15.2).
            _statusPend := FALSE;
        ELSE
            // A command the controller never acknowledged: its own first-out, which
            // the robot CM adopts verbatim (§8.2).
            _lastResult.ReasonCode  := PL_TcpDevReasons.DEV_RESP_TIMEOUT;
            _lastResult.Description := 'std.error.deviceResponseTimeout';
            _lastResult.SourcePath  := Name;
            _busy := FALSE;
        END_IF
    E_AsciiLinkEvent.OVERFLOW:
        _M_Lost(Reason := E_Reason.DEVICE_PROTOCOL_ERROR, Text := 'std.error.deviceResponseOverflow');
    E_AsciiLinkEvent.CHANNEL_FAULT:
        _M_Lost(Reason := E_Reason.LINK_TIMEOUT, Text := 'std.error.transportChannelFault');
ELSE
    _M_Lost(Reason := E_Reason.DEVICE_PROTOCOL_ERROR, Text := 'std.error.byteChannelStateInvalid');
END_CASE
// The peer closed the socket: the session is gone now, not after a timeout.
IF _sessionUp AND (LinkState = E_ByteChannelState.CLOSED) THEN
    _M_Lost(Reason := E_Reason.LINK_TIMEOUT, Text := 'std.error.robotLinkDown');
END_IF
Cyclic := SUPER^.Cyclic();
// A lost link invalidates every cached fact. Publishing a stale pose or a stale
// "not in protective stop" while disconnected would be worse than publishing
// nothing, because both read as positive statements about a robot we cannot see.
IF NOT Linked THEN
    _busy       := FALSE;
    _referenced := FALSE;
    _mode       := E_RobotOpMode.UNKNOWN;
    _area       := 0;
    _resumable  := FALSE;
END_IF
END_METHOD

METHOD PROTECTED _M_Open : BOOL
_statusPend := FALSE;
_hbReply := FALSE;
_M_Open := _link.M_Open(Host := ParCfg.Host, Port := ParCfg.Port);
END_METHOD

METHOD PROTECTED _M_Close : BOOL
_link.M_Close();
_statusPend := FALSE;
_busy := FALSE;
_M_Close := TRUE;
END_METHOD

// The heartbeat IS the status poll. With a command reply still outstanding the
// slot is taken, so that reply is awaited instead: any well-formed reply proves the
// controller alive, and the one-outstanding-request rule is never broken by
// housekeeping.
METHOD PROTECTED _M_HbStart : BOOL
_hbReply := FALSE;
IF _link.Pending THEN
    _M_HbStart := TRUE;
    RETURN;
END_IF
_M_HbStart := _link.M_Send(Text := 'STA');
_statusPend := _M_HbStart;
END_METHOD

METHOD PROTECTED _M_HbPoll : E_HbResult
IF _hbReply THEN
    _M_HbPoll := E_HbResult.OK;
ELSE
    _M_HbPoll := E_HbResult.PENDING;   // silence is judged by LinkTimeout in the base
END_IF
END_METHOD

// Parse one terminated reply. Status replies refresh the published facts; command
// replies clear Busy or record the controller's own first-out.
METHOD PROTECTED _M_OnResponse
VAR_INPUT
    Response : STRING(255);
END_VAR
VAR
    _cmd  : STRING(16);
    _stat : STRING(16);
END_VAR
// Any well-formed reply is evidence the controller is alive (§3.15.2).
_hbReply := TRUE;

_cmd  := _M_Field(Response, 1);
_stat := _M_Field(Response, 2);

IF _stat = 'ERR' THEN
    // The controller refused or faulted. Carry ITS message verbatim rather than a
    // paraphrase - a service technician needs the robot's own text (S8.2). The
    // robot CM adopts it from LastResult as its first-out.
    _ctrlMsg := _M_MakeCtrlDiag(Code := _M_Field(Response, 3),
                                Text := _M_Field(Response, 4));
    _lastResult := _ctrlMsg;
    _busy := FALSE;
    _statusPend := FALSE;
    RETURN;
END_IF

IF _cmd = 'STA' THEN
    // STA,OK,<busy>,<ref>,<mode>,<area>,<prot>,<resumable>,<x>,<y>,<z>,<rx>,<ry>,<rz>
    _busy       := (_M_Field(Response, 3) = '1');
    _referenced := (_M_Field(Response, 4) = '1');
    _mode       := _M_ToMode(_M_Field(Response, 5));
    _area       := DINT_TO_DWORD(STRING_TO_DINT(_M_Field(Response, 6)));
    _protStop   := (_M_Field(Response, 7) = '1');
    _resumable  := (_M_Field(Response, 8) = '1');
    _pose.X     := STRING_TO_LREAL(_M_Field(Response, 9));
    _pose.Y     := STRING_TO_LREAL(_M_Field(Response, 10));
    _pose.Z     := STRING_TO_LREAL(_M_Field(Response, 11));
    _pose.RX    := STRING_TO_LREAL(_M_Field(Response, 12));
    _pose.RY    := STRING_TO_LREAL(_M_Field(Response, 13));
    _pose.RZ    := STRING_TO_LREAL(_M_Field(Response, 14));
    _statusPend := FALSE;
    RETURN;
END_IF

// A command reply. The robot has ACCEPTED it; completion is observed through the
// status poll, so a long path does not hold the request slot for its duration.
_statusPend := FALSE;
END_METHOD

// Issue one ID-addressed request. FALSE = refused outright, with LastResult set,
// which is what the CM turns into a first-out (S5.6).
METHOD PRIVATE _M_Request : BOOL
VAR_INPUT
    Text : STRING(255);
END_VAR
_M_Request := FALSE;
IF NOT Linked THEN
    _lastResult := _M_MakeLinkDiag();
    RETURN;
END_IF
IF _link.Pending THEN
    // One outstanding request is the link's rule; refusing here keeps the caller
    // honest instead of silently dropping the command.
    _lastResult := _M_MakeLinkDiag();
    RETURN;
END_IF
IF NOT _link.M_Send(Text := Text) THEN
    _lastResult := _M_MakeLinkDiag();
    RETURN;
END_IF
_statusPend := FALSE;
_busy := TRUE;
_M_Request := TRUE;
END_METHOD

// n-th comma-separated field of a response, 1-based; '' when absent. Bounded and
// allocation-free (O10).
METHOD PRIVATE _M_Field : STRING(64)
VAR_INPUT
    Text : STRING(255);
    N    : INT;
END_VAR
VAR
    i, count, start, len_ : INT;
    ch : STRING(1);
END_VAR
_M_Field := '';
count := 1;
start := 1;
len_ := LEN(Text);
FOR i := 1 TO len_ DO
    ch := MID(Text, 1, i);
    IF ch = ',' THEN
        IF count = N THEN
            _M_Field := MID(Text, i - start, start);
            RETURN;
        END_IF
        count := count + 1;
        start := i + 1;
    END_IF
END_FOR
IF count = N THEN
    _M_Field := MID(Text, len_ - start + 1, start);
END_IF
END_METHOD

// Controller mode text -> E_RobotOpMode. Anything unrecognised is UNKNOWN, never
// a permissive mode: an unparsed reply must not read as "auto is granted".
METHOD PRIVATE _M_ToMode : E_RobotOpMode
VAR_INPUT
    ModeText : STRING(64);
END_VAR
IF ModeText = 'AUTO' THEN
    _M_ToMode := E_RobotOpMode.AUTO_REMOTE;
ELSIF ModeText = 'MANR' THEN
    _M_ToMode := E_RobotOpMode.MANUAL_REDUCED;
ELSIF ModeText = 'MANH' THEN
    _M_ToMode := E_RobotOpMode.MANUAL_HIGH;
ELSE
    _M_ToMode := E_RobotOpMode.UNKNOWN;
END_IF
END_METHOD

// Wrap the controller's own error into a Fraktal diagnostic without translating it.
METHOD PRIVATE _M_MakeCtrlDiag : ST_Diagnostic
VAR_INPUT
    Code : STRING(64);
    Text : STRING(64);
END_VAR
_M_MakeCtrlDiag.ReasonCode  := PL_ModuleReasons.ROBOT_CONTROLLER_FAULT;
_M_MakeCtrlDiag.Description := CONCAT(CONCAT(Code, ' '), Text);
_M_MakeCtrlDiag.SourcePath  := Name;
END_METHOD

// The link is the reason a request was refused; reuse the Framework band rather
// than minting a robot code for a transport fact (Annex D).
METHOD PRIVATE _M_MakeLinkDiag : ST_Diagnostic
_M_MakeLinkDiag.ReasonCode  := E_Reason.LINK_TIMEOUT;
_M_MakeLinkDiag.Description := 'std.error.robotLinkDown';
_M_MakeLinkDiag.SourcePath  := Name;
END_METHOD

METHOD PowerOn : BOOL
PowerOn := _M_Request('PWR,1');
END_METHOD

METHOD PowerOff : BOOL
PowerOff := _M_Request('PWR,0');
END_METHOD

METHOD Home : BOOL
Home := _M_Request('HOME');
END_METHOD

METHOD MoveToPoint : BOOL
VAR_INPUT
    PointId : DWORD;
END_VAR
MoveToPoint := _M_Request(CONCAT('MOV,', DWORD_TO_STRING(PointId)));
END_METHOD

METHOD RunPath : BOOL
VAR_INPUT
    ListId   : DWORD;
    StartIdx : DINT;
    EndIdx   : DINT;
END_VAR
RunPath := _M_Request(CONCAT(CONCAT(CONCAT(CONCAT(CONCAT(
    'PTH,', DWORD_TO_STRING(ListId)), ','), DINT_TO_STRING(StartIdx)), ','),
    DINT_TO_STRING(EndIdx)));
END_METHOD

METHOD Interrupt : BOOL
Interrupt := _M_Request('INT');
END_METHOD

METHOD Resume : BOOL
// Refuse rather than execute when the arm has left the retained path (I.4b).
IF NOT _resumable THEN
    Resume := FALSE;
    RETURN;
END_IF
Resume := _M_Request('RES');
END_METHOD

METHOD Abort : BOOL
Abort := _M_Request('ABT');
_busy := FALSE;
END_METHOD

METHOD ResetController : BOOL
ResetController := _M_Request('RST');
END_METHOD

METHOD RequestMode : BOOL
VAR_INPUT
    Mode : E_RobotOpMode;
END_VAR
VAR
    _s : STRING(8);
END_VAR
CASE Mode OF
    E_RobotOpMode.AUTO_REMOTE:    _s := 'AUTO';
    E_RobotOpMode.MANUAL_REDUCED: _s := 'MANR';
    E_RobotOpMode.MANUAL_HIGH:    _s := 'MANH';
ELSE
    // Requesting UNKNOWN is meaningless and must not reach the controller.
    RequestMode := FALSE;
    RETURN;
END_CASE
// Record what we ASKED for. ActualMode stays whatever the controller reports, so
// an ungranted request stays visibly ungranted (I.4a(a)).
_reqMode := Mode;
RequestMode := _M_Request(CONCAT('MOD,', _s));
END_METHOD

METHOD SetTool : BOOL
VAR_INPUT
    ToolId : DWORD;
END_VAR
SetTool := _M_Request(CONCAT('TOO,', DWORD_TO_STRING(ToolId)));
END_METHOD

METHOD SetFrame : BOOL
VAR_INPUT
    FrameId : DWORD;
END_VAR
SetFrame := _M_Request(CONCAT('FRM,', DWORD_TO_STRING(FrameId)));
END_METHOD

METHOD SetPayload : BOOL
VAR_INPUT
    LoadId : DWORD;
END_VAR
SetPayload := _M_Request(CONCAT('PLD,', DWORD_TO_STRING(LoadId)));
END_METHOD

METHOD Jog : BOOL
VAR_INPUT
    Mode : E_RobotJogMode;
    Axis : INT;
    Dir  : INT;
END_VAR
// Jogging requires a manual mode on the CONTROLLER, not merely a PLC release:
// the mode is what physically bounds the motion (I.4a(a)).
IF (_mode <> E_RobotOpMode.MANUAL_REDUCED) AND (_mode <> E_RobotOpMode.MANUAL_HIGH) THEN
    Jog := FALSE;
    RETURN;
END_IF
Jog := _M_Request(CONCAT(CONCAT(CONCAT(CONCAT(CONCAT(
    'JOG,', DINT_TO_STRING(Mode)), ','), INT_TO_STRING(Axis)), ','),
    INT_TO_STRING(Dir)));
END_METHOD

METHOD RunPallet : BOOL
VAR_INPUT
    PalletId : DWORD;
    Nest     : DINT;
END_VAR
RunPallet := _M_Request(CONCAT(CONCAT(CONCAT(
    'PAL,', DWORD_TO_STRING(PalletId)), ','), DINT_TO_STRING(Nest)));
END_METHOD

METHOD MoveTemplate : BOOL
VAR_INPUT
    FromPosId : DWORD;
    ToPosId   : DWORD;
END_VAR
MoveTemplate := _M_Request(CONCAT(CONCAT(CONCAT(
    'TPL,', DWORD_TO_STRING(FromPosId)), ','), DWORD_TO_STRING(ToPosId)));
END_METHOD

METHOD MoveFromArea : BOOL
VAR_INPUT
    ToPosId : DWORD;
END_VAR
MoveFromArea := _M_Request(CONCAT('ARE,', DWORD_TO_STRING(ToPosId)));
END_METHOD

METHOD SetSpeedScale : BOOL
VAR_INPUT
    Percent : REAL;
END_VAR
IF (Percent < 0.0) OR (Percent > 100.0) THEN
    SetSpeedScale := FALSE;
    RETURN;
END_IF
SetSpeedScale := _M_Request(CONCAT('SPD,', REAL_TO_STRING(Percent)));
END_METHOD

// The ROBOT is moving. The base already owns Busy for its own command handshake;
// conflating the two would make "is the arm moving" unanswerable.
PROPERTY MotionBusy : BOOL
GET
MotionBusy := _busy;
END_GET
END_PROPERTY

PROPERTY Referenced : BOOL
GET
Referenced := _referenced;
END_GET
END_PROPERTY

PROPERTY ActualMode : E_RobotOpMode
GET
ActualMode := _mode;
END_GET
END_PROPERTY

PROPERTY ActualPosition : ST_RobotPose
GET
ActualPosition := _pose;
END_GET
END_PROPERTY

PROPERTY ControllerMessage : ST_Diagnostic
GET
ControllerMessage := _ctrlMsg;
END_GET
END_PROPERTY

PROPERTY CurrentArea : DWORD
GET
CurrentArea := _area;
END_GET
END_PROPERTY

PROPERTY ProtectiveStop : BOOL
GET
ProtectiveStop := _protStop;
END_GET
END_PROPERTY

PROPERTY Resumable : BOOL
GET
Resumable := _resumable;
END_GET
END_PROPERTY

PROPERTY LastResult : ST_Diagnostic
GET
LastResult := _lastResult;
END_GET
END_PROPERTY

END_FUNCTION_BLOCK

// ---- FB_RobotRoutePlanner.TcPOU
// Annex I I.9-I.10.2 / Core S10.7 - the generic route planner.
//
// The station supplies a route graph and taught geometry as CONFIGURATION and
// writes no traversal code. This type resolves, for any pair of positions:
//
//     from -> departHelp -> (help-graph search) -> approachHelp -> to
//
// and emits the resulting bounded point list. It is pure logic: no I/O, no
// connector, no motion. That is deliberate - it makes the part of the robot
// layer that is genuinely Fraktal's own testable against a fixture with no arm
// (S5.7, Annex H), which is why it is built first.
//
// Positions are indices, not enum values: the application's HELPn / nest enums
// map onto 1..MAX_HELPS and 1..MAX_NESTS. 0 means "not this kind of position",
// so exactly one of Nest/Help is non-zero at each end of a move.
FUNCTION_BLOCK FB_RobotRoutePlanner
VAR_INPUT
    {attribute 'OPC.UA.DA' := '0'}
    rGraph : REFERENCE TO ST_RouteGraph;
    {attribute 'OPC.UA.DA' := '0'}
    rGeom  : REFERENCE TO ST_RobotGeometry;
END_VAR
VAR
    // bounded breadth-first search over the help graph; no allocation (O10)
    _seen  : ARRAY[1..PL_RobotPlanner.MAX_HELPS] OF BOOL;
    _prev  : ARRAY[1..PL_RobotPlanner.MAX_HELPS] OF INT;
    _queue : ARRAY[1..PL_RobotPlanner.MAX_HELPS] OF INT;
    _chain : ARRAY[1..PL_RobotPlanner.MAX_HELPS] OF INT;
    _chainCount : INT;
    _overflow   : BOOL;   // a route longer than MAX_ROUTE_POINTS was attempted
END_VAR

// Nothing cyclic: the planner is called on demand.
;

// Plan a move and emit its point list. Returns 0 on success, or the S8.8 reason
// the caller should fault with - the planner never raises events itself, so it
// stays usable from a test with no module around it.
METHOD PUBLIC BuildRoute : DINT
VAR_INPUT
    Gripper  : INT;
    FromNest : INT;   // 0 = start is a help position
    FromHelp : INT;   // 0 = start is a nest
    ToNest   : INT;   // 0 = target is a help position
    ToHelp   : INT;   // 0 = target is a nest
END_VAR
VAR_IN_OUT
    Route : ST_RobotPointList;
END_VAR
VAR
    _departHelp   : INT;
    _approachHelp : INT;
    _direct       : DWORD;
    _i            : INT;
END_VAR
Route.Count := 0;
_overflow := FALSE;
BuildRoute := 0;

IF NOT __ISVALIDREF(rGraph) OR NOT __ISVALIDREF(rGeom) THEN
    BuildRoute := PL_ModuleReasons.ROBOT_NO_ROUTE;
    RETURN;
END_IF
IF NOT _M_ValidEnds(Gripper, FromNest, FromHelp, ToNest, ToHelp) THEN
    BuildRoute := PL_ModuleReasons.ROBOT_NO_ROUTE;
    RETURN;
END_IF

// A taught nest -> nest list bypasses help routing entirely (I.9 DirectNest).
IF (FromNest <> 0) AND (ToNest <> 0) THEN
    _direct := rGraph.DirectNest[FromNest, ToNest];
    IF _direct <> 0 THEN
        _M_AddList(_direct, Route);
        IF _overflow THEN BuildRoute := PL_ModuleReasons.ROBOT_NO_ROUTE; END_IF
        RETURN;
    END_IF
END_IF

// Leaving a nest: resolve the corridor out, then emit it (nest-ward -> help-ward).
_departHelp := FromHelp;
IF FromNest <> 0 THEN
    _departHelp := ResolveHelp(Gripper := Gripper, Nest := FromNest,
        OtherRegion := _M_RegionOf(Gripper, ToNest, ToHelp), Dir := E_HelpRole.DEPART);
    IF _departHelp = 0 THEN
        BuildRoute := PL_ModuleReasons.ROBOT_NO_HELP_FOR_NEST;
        RETURN;
    END_IF
    _M_EmitCorridor(Gripper, FromNest, _departHelp, E_HelpRole.DEPART, Route);
END_IF

// Entering a nest: resolve the corridor in BEFORE searching, so an unroutable
// nest is reported as such rather than as a missing help-graph edge (S5.6).
_approachHelp := ToHelp;
IF ToNest <> 0 THEN
    _approachHelp := ResolveHelp(Gripper := Gripper, Nest := ToNest,
        OtherRegion := _M_RegionOf(Gripper, FromNest, FromHelp), Dir := E_HelpRole.APPROACH);
    IF _approachHelp = 0 THEN
        BuildRoute := PL_ModuleReasons.ROBOT_NO_HELP_FOR_NEST;
        RETURN;
    END_IF
END_IF

// The transit itself.
IF NOT _M_FindHelpChain(_departHelp, _approachHelp) THEN
    BuildRoute := PL_ModuleReasons.ROBOT_NO_ROUTE;
    RETURN;
END_IF
FOR _i := 1 TO _chainCount DO
    _M_AddPose(rGeom.HelpPose[_chain[_i]], E_MoveClass.FAST_PTP, Route);
END_FOR

// Arriving: the approach corridor reversed, ending exactly on the nest.
IF ToNest <> 0 THEN
    _M_EmitCorridor(Gripper, ToNest, _approachHelp, E_HelpRole.APPROACH, Route);
END_IF

IF _overflow THEN
    Route.Count := 0;
    BuildRoute := PL_ModuleReasons.ROBOT_NO_ROUTE;
END_IF
END_METHOD

// Which help serves this nest for this direction of travel. Role-primary:
// direction is the higher-consequence constraint, because a wrong-direction
// corridor can drive the tool into the fixture while a wrong region is only a
// longer, still-safe route. Region breaks ties among same-direction corridors.
// Returns 0 when no corridor is legal - a one-way nest asked to reverse.
METHOD PUBLIC ResolveHelp : INT
VAR_INPUT
    Gripper     : INT;
    Nest        : INT;
    OtherRegion : DWORD;
    Dir         : E_HelpRole;
END_VAR
VAR
    _i     : INT;
    _n     : INT;
    _cand  : ARRAY[1..PL_RobotPlanner.MAX_HELPS_PER_NEST] OF INT;
    _first : INT;
END_VAR
ResolveHelp := 0;
IF NOT __ISVALIDREF(rGraph) THEN RETURN; END_IF
IF (Gripper < 1) OR (Gripper > PL_RobotPlanner.MAX_GRIPPERS) THEN RETURN; END_IF
IF (Nest < 1) OR (Nest > PL_RobotPlanner.MAX_NESTS) THEN RETURN; END_IF

// 1) VALIDITY FILTER - keep only corridors legal for this direction.
//    EITHER is always legal, so a nest is exit-able the way it was entered
//    unless its geometry is declared physically one-way.
_n := 0;
FOR _i := 1 TO rGraph.NestHelp[Gripper, Nest].Count DO
    IF rGraph.NestHelp[Gripper, Nest].Helps[_i].HelpId <> 0 THEN
        IF (rGraph.NestHelp[Gripper, Nest].Helps[_i].Role = Dir)
        OR (rGraph.NestHelp[Gripper, Nest].Helps[_i].Role = E_HelpRole.EITHER) THEN
            _n := _n + 1;
            _cand[_n] := _i;
        END_IF
    END_IF
END_FOR

IF _n = 0 THEN RETURN; END_IF
IF _n = 1 THEN
    ResolveHelp := rGraph.NestHelp[Gripper, Nest].Helps[_cand[1]].HelpId;
    RETURN;
END_IF

// 2) TIE-BREAK - among same-direction corridors prefer the one whose region
//    matches the other endpoint's side; otherwise the first candidate. Region
//    configuration is therefore needed ONLY on a nest with two corridors for
//    the same direction.
_first := rGraph.NestHelp[Gripper, Nest].Helps[_cand[1]].HelpId;
FOR _i := 1 TO _n DO
    IF (OtherRegion <> 0)
    AND (rGraph.NestHelp[Gripper, Nest].Helps[_cand[_i]].RegionId = OtherRegion) THEN
        ResolveHelp := rGraph.NestHelp[Gripper, Nest].Helps[_cand[_i]].HelpId;
        RETURN;
    END_IF
END_FOR
ResolveHelp := _first;
END_METHOD

// Breadth-first search over the help adjacency, filling _chain / _chainCount
// with the help sequence from a to b inclusive. Bounded and allocation-free.
METHOD PRIVATE _M_FindHelpChain : BOOL
VAR_INPUT
    HelpFrom : INT;
    HelpTo   : INT;
END_VAR
VAR
    _head : INT;
    _tail : INT;
    _cur  : INT;
    _nxt  : INT;
    _i    : INT;
    _walk : INT;
END_VAR
_M_FindHelpChain := FALSE;
_chainCount := 0;
IF (HelpFrom < 1) OR (HelpFrom > PL_RobotPlanner.MAX_HELPS) THEN RETURN; END_IF
IF (HelpTo   < 1) OR (HelpTo   > PL_RobotPlanner.MAX_HELPS) THEN RETURN; END_IF

IF HelpFrom = HelpTo THEN
    _chain[1] := HelpFrom;
    _chainCount := 1;
    _M_FindHelpChain := TRUE;
    RETURN;
END_IF

FOR _i := 1 TO PL_RobotPlanner.MAX_HELPS DO
    _seen[_i] := FALSE;
    _prev[_i] := 0;
END_FOR

_head := 1;
_tail := 1;
_queue[1] := HelpFrom;
_seen[HelpFrom] := TRUE;

WHILE _head <= _tail DO
    _cur := _queue[_head];
    _head := _head + 1;
    FOR _nxt := 1 TO PL_RobotPlanner.MAX_HELPS DO
        IF rGraph.HelpAdj[_cur, _nxt] AND NOT _seen[_nxt] THEN
            _seen[_nxt] := TRUE;
            _prev[_nxt] := _cur;
            IF _nxt = HelpTo THEN
                // walk the predecessors back, then reverse into _chain
                _walk := HelpTo;
                _chainCount := 0;
                WHILE _walk <> 0 DO
                    _chainCount := _chainCount + 1;
                    _queue[_chainCount] := _walk;
                    _walk := _prev[_walk];
                END_WHILE
                FOR _i := 1 TO _chainCount DO
                    _chain[_i] := _queue[_chainCount - _i + 1];
                END_FOR
                _M_FindHelpChain := TRUE;
                RETURN;
            END_IF
            _tail := _tail + 1;
            _queue[_tail] := _nxt;
        END_IF
    END_FOR
END_WHILE
END_METHOD

// Emit one corridor. DEPART runs the steps nest-ward -> help-ward, leaving the
// arm heading out; APPROACH runs them reversed and then lands exactly on the
// nest. They are separate definitions, not one another reversed, so a
// lift-then-clear retract can differ from a straight-in approach (I.10.1).
METHOD PRIVATE _M_EmitCorridor
VAR_INPUT
    Gripper : INT;
    Nest    : INT;
    HelpId  : INT;
    Dir     : E_HelpRole;
END_VAR
VAR_IN_OUT
    Route : ST_RobotPointList;
END_VAR
VAR
    _i   : INT;
    _idx : INT;
    _c   : ST_Corridor;
END_VAR
_idx := _M_AffinityIndex(Gripper, Nest, HelpId);
IF _idx = 0 THEN RETURN; END_IF

IF Dir = E_HelpRole.DEPART THEN
    _c := rGraph.NestHelp[Gripper, Nest].Helps[_idx].Depart;
ELSE
    _c := rGraph.NestHelp[Gripper, Nest].Helps[_idx].Approach;
END_IF

// A taught corridor: one point naming the list, for the executor to run here.
IF (_c.StepCount = 0) AND (_c.ListId <> 0) THEN
    _M_AddList(_c.ListId, Route);
    RETURN;
END_IF

IF Dir = E_HelpRole.DEPART THEN
    FOR _i := 1 TO _c.StepCount DO
        _M_AddPose(_M_Offset(rGeom.NestPose[Gripper, Nest], _c.Steps[_i].D),
                   _c.Steps[_i].MoveClass, Route);
    END_FOR
ELSE
    FOR _i := _c.StepCount TO 1 BY -1 DO
        _M_AddPose(_M_Offset(rGeom.NestPose[Gripper, Nest], _c.Steps[_i].D),
                   _c.Steps[_i].MoveClass, Route);
    END_FOR
    // and finally the nest itself, reached exactly (I.8 last-point-exact)
    _M_AddPose(rGeom.NestPose[Gripper, Nest], E_MoveClass.SLOW_LINEAR, Route);
END_IF
END_METHOD

// Index of the affinity entry naming this help on this nest; 0 if absent.
METHOD PRIVATE _M_AffinityIndex : INT
VAR_INPUT
    Gripper : INT;
    Nest    : INT;
    HelpId  : INT;
END_VAR
VAR
    _i : INT;
END_VAR
_M_AffinityIndex := 0;
FOR _i := 1 TO rGraph.NestHelp[Gripper, Nest].Count DO
    IF rGraph.NestHelp[Gripper, Nest].Helps[_i].HelpId = HelpId THEN
        _M_AffinityIndex := _i;
        RETURN;
    END_IF
END_FOR
END_METHOD

// The transit region of the move's other endpoint, used only to break ties
// between same-direction corridors. A help carries its region directly; a nest
// borrows the region of its first serving help.
METHOD PRIVATE _M_RegionOf : DWORD
VAR_INPUT
    Gripper : INT;
    Nest    : INT;
    Help    : INT;
END_VAR
VAR
    _h : INT;
END_VAR
_M_RegionOf := 0;
IF (Help >= 1) AND (Help <= PL_RobotPlanner.MAX_HELPS) THEN
    _M_RegionOf := rGraph.HelpRegion[Help];
    RETURN;
END_IF
IF (Nest >= 1) AND (Nest <= PL_RobotPlanner.MAX_NESTS)
AND (Gripper >= 1) AND (Gripper <= PL_RobotPlanner.MAX_GRIPPERS) THEN
    IF rGraph.NestHelp[Gripper, Nest].Count >= 1 THEN
        _h := rGraph.NestHelp[Gripper, Nest].Helps[1].HelpId;
        IF (_h >= 1) AND (_h <= PL_RobotPlanner.MAX_HELPS) THEN
            _M_RegionOf := rGraph.HelpRegion[_h];
        END_IF
    END_IF
END_IF
END_METHOD

// Pose + offset, in the nest's own frame. This is a corridor step, not a
// general transform - chained frames are the connector's job (I.12).
METHOD PRIVATE _M_Offset : ST_RobotPose
VAR_INPUT
    Base : ST_RobotPose;
    D    : ST_RobotPose;
END_VAR
_M_Offset.X  := Base.X  + D.X;
_M_Offset.Y  := Base.Y  + D.Y;
_M_Offset.Z  := Base.Z  + D.Z;
_M_Offset.RX := Base.RX + D.RX;
_M_Offset.RY := Base.RY + D.RY;
_M_Offset.RZ := Base.RZ + D.RZ;
END_METHOD

// Append a move-to-pose point, refusing rather than growing past the bound.
METHOD PRIVATE _M_AddPose
VAR_INPUT
    P  : ST_RobotPose;
    MC : E_MoveClass;
END_VAR
VAR_IN_OUT
    Route : ST_RobotPointList;
END_VAR
IF Route.Count >= PL_RobotPlanner.MAX_ROUTE_POINTS THEN
    _overflow := TRUE;
    RETURN;
END_IF
Route.Count := Route.Count + 1;
Route.Points[Route.Count].Target    := P;
Route.Points[Route.Count].MoveClass := MC;
Route.Points[Route.Count].ListId    := 0;
END_METHOD

// Append a run-this-taught-list point.
METHOD PRIVATE _M_AddList
VAR_INPUT
    ListId : DWORD;
END_VAR
VAR_IN_OUT
    Route : ST_RobotPointList;
END_VAR
IF Route.Count >= PL_RobotPlanner.MAX_ROUTE_POINTS THEN
    _overflow := TRUE;
    RETURN;
END_IF
Route.Count := Route.Count + 1;
Route.Points[Route.Count].ListId := ListId;
END_METHOD

// Exactly one of Nest/Help at each end, and every index in range (S5.6).
METHOD PRIVATE _M_ValidEnds : BOOL
VAR_INPUT
    Gripper  : INT;
    FromNest : INT;
    FromHelp : INT;
    ToNest   : INT;
    ToHelp   : INT;
END_VAR
_M_ValidEnds := FALSE;
IF (Gripper < 1) OR (Gripper > PL_RobotPlanner.MAX_GRIPPERS) THEN RETURN; END_IF
IF (FromNest = 0) = (FromHelp = 0) THEN RETURN; END_IF
IF (ToNest   = 0) = (ToHelp   = 0) THEN RETURN; END_IF
IF (FromNest < 0) OR (FromNest > PL_RobotPlanner.MAX_NESTS) THEN RETURN; END_IF
IF (ToNest   < 0) OR (ToNest   > PL_RobotPlanner.MAX_NESTS) THEN RETURN; END_IF
IF (FromHelp < 0) OR (FromHelp > PL_RobotPlanner.MAX_HELPS) THEN RETURN; END_IF
IF (ToHelp   < 0) OR (ToHelp   > PL_RobotPlanner.MAX_HELPS) THEN RETURN; END_IF
_M_ValidEnds := TRUE;
END_METHOD

END_FUNCTION_BLOCK

// ---- FB_RobotCM.TcPOU
// Annex I I.4 - the robot Control Module. An ordinary CM: it EXTENDS
// FB_ControlModuleBase and adds only its device logic; the handshake, first-out
// stamping, rollup and publication are base-owned and proven in FB_Base_Tests.
//
// Its additions over a plain CM are the annex's three device facts plus the
// HELD translation:
//   - every command first requires Linked (Annex D), and a refusal is ADOPTED
//     verbatim from the connector's LastResult rather than re-classified (S8.2);
//   - validate-then-command (S5.6): the speed band, the controller's reported
//     mode and the reference state are checked BEFORE anything reaches the floor,
//     in that order - a bad parameter is malformed regardless of the mode, and
//     a mode problem is more specific than a reference problem;
//   - a protective stop aborts with its OWN reason so the alarm record never
//     misreports a process event as a safety event (I.4a(c));
//   - a lost permissive HOLDS on-path (I.4b): the connector is Interrupted at
//     hold onset and Resumed on release, and a release that cannot resume -
//     the arm was jogged while held - faults ROBOT_RESUME_INVALID instead of
//     driving back through untaught space. HELD, not fault, for the permissive
//     itself: that is this repo's settled doctrine (a lost permissive is
//     restorable operator/process state, Core S6.1).
//
// NOT yet raised here: ROBOT_SAFETY_DROPPED. Safety status is S9 read-only and
// nothing feeds this type a safety alias yet; the reason lands with the code
// that raises it.
FUNCTION_BLOCK FB_RobotCM EXTENDS FB_ControlModuleBase
VAR_INPUT
    Command : E_RobotCommand;
    ParCfg  : ST_RobotParCfg;
    ParCmd  : ST_RobotParCmd;
END_VAR
VAR_OUTPUT
    OutCmd : ST_RobotOutCmd;
    OutImm : ST_RobotOutImm;
    Intlk  : FB_PermIntlk;   // conditions are DECLARED BY THE APPLICATION (S7.2)
END_VAR
VAR
    {attribute 'OPC.UA.DA' := '0'}
    _conn        : I_RobotConnector;
    _tMove       : TON;
    _heldOnPath  : BOOL;                 // an Interrupt is outstanding (I.4b)
    _startResult : ST_Diagnostic;        // connector LastResult at command start
    _appCond     : ARRAY[1..PL_Fraktal.MAX_PERMINTLK_COND] OF BOOL;
END_VAR

Cyclic();

// Wire identity and the connector. Called once from the owning EM/Unit (S3.11).
METHOD Setup : BOOL
VAR_INPUT
    Name  : STRING(80);
    Robot : I_RobotConnector;
END_VAR
_M_SetName(Name);
_M_SetPresentation(DisplayNameKey := 'std.moduleType.robot.name', DescriptionKey := 'std.moduleType.robot.description', TypeKey := 'std.moduleType.robot');
IF Robot = 0 THEN
    _M_Fault(E_Reason.UNSUPPORTED_COMMAND, 'std.error.robotLinkDown');
    Setup := FALSE;
    RETURN;
END_IF
_conn := Robot;
Setup := TRUE;
END_METHOD

// S3.14 one-shot on the accepted Execute edge, before OnCyclic/_M_Dispatch.
// Command-local reset only - the process behaviour stays in dispatch.
METHOD PROTECTED OnCommandStart : DINT
OnCommandStart := SUPER^.OnCommandStart();
OutCmd.ReachedId := 0;
_heldOnPath      := FALSE;
_tMove(IN := FALSE);
// The connector's reason at command start. Everything after this is compared
// against it, so an OLD fault is never re-adopted as if this command caused it.
IF _conn <> 0 THEN
    _startResult := _conn.LastResult;
END_IF
END_METHOD

// Mirror the connector's published facts; the device logic is in _M_Dispatch.
METHOD PROTECTED OnCyclic : DINT
VAR
    _c : ST_Diagnostic;
END_VAR
OnCyclic := SUPER^.OnCyclic();

IF _conn <> 0 THEN
    // §3.15.3 - the CM services its connector every scan, so session, heartbeat
    // and reconnect stay live whichever connector is wired; a project ticks nothing.
    _conn.Cyclic();
    OutImm.Linked         := _conn.Linked;
    OutImm.Referenced     := _conn.Referenced;
    OutImm.MotionBusy     := _conn.MotionBusy;
    OutImm.ActualMode     := _conn.ActualMode;
    OutImm.CurrentArea    := _conn.CurrentArea;
    OutImm.ProtectiveStop := _conn.ProtectiveStop;
    OutImm.Resumable      := _conn.Resumable;
    OutImm.SpeedScale     := ParCmd.SpeedScale;
ELSE
    // No connector wired: every published fact is FALSE/0 rather than stale.
    OutImm.Linked         := FALSE;
    OutImm.Referenced     := FALSE;
    OutImm.MotionBusy     := FALSE;
    OutImm.ActualMode     := E_RobotOpMode.UNKNOWN;
    OutImm.CurrentArea    := 0;
    OutImm.ProtectiveStop := FALSE;
    OutImm.Resumable      := FALSE;
END_IF
END_METHOD

// The ONLY thing this type writes (Core S2.2): validation ladder (S5.6), then the
// ID-addressed primitive, then completion/hold/timeout at step 20.
METHOD PROTECTED _M_Dispatch
VAR
    _scale : REAL;
    _cd    : ST_Diagnostic;   // C0185: cannot read .member off a property result
END_VAR
// ---- validation BEFORE motion (S5.6) --------------------------------------
// Order is deliberate: a malformed parameter is wrong regardless of mode, and a
// mode problem is more specific than a reference problem - so each rejection
// sends the operator to the real cause rather than the first one checked.
IF _conn = 0 THEN
    _M_Fault(E_Reason.LINK_TIMEOUT, 'std.error.robotLinkDown');
    RETURN;
END_IF
// §3.15.4 - the deliberate reconnect. It stays BUSY until the link is back (the
// Unit's stall guard names it if it never is) and resumes nothing (§3.15.2):
// clearing the robot's own fault is part of it only when asked for.
IF Command = E_RobotCommand.RECONNECT THEN
    _M_Tag();
    IF NOT _conn.Linked THEN
        _conn.Connect();
        RETURN;
    END_IF
    IF ParCmd.AcknowledgeController THEN
        _conn.ResetController();
    END_IF
    _M_Complete();
    RETURN;
END_IF
IF NOT _conn.Linked THEN
    _M_Fault(E_Reason.LINK_TIMEOUT, 'std.error.robotLinkDown');
    RETURN;
END_IF
_M_Tag();
_M_ApplyConditions();
IF _M_IsMotion(Command) THEN
    IF (ParCmd.SpeedScale < ParCfg.SpeedScaleMin) OR (ParCmd.SpeedScale > ParCfg.SpeedScaleMax) THEN
        _M_FaultN(Code := PL_ModuleReasons.ROBOT_PARAM_OOR, Text := 'std.error.robotSpeedScaleOutOfRange');
        RETURN;
    END_IF
    // The controller REPORTED mode bounds what motion is physically allowed; an
    // unreported (UNKNOWN) mode is never treated as permissive (I.4a(a)).
    IF _conn.ActualMode <> E_RobotOpMode.AUTO_REMOTE THEN
        _M_FaultN(Code := PL_ModuleReasons.ROBOT_MODE_NOT_PERMITTED, Text := 'std.error.robotModeNotPermitted');
        RETURN;
    END_IF
    // HOME is deliberately exempt: homing is what ESTABLISHES the reference, so
    // requiring one first would make the robot permanently unhomeable - the
    // deadlock this ladder exists to prevent, not create.
    IF (Command <> E_RobotCommand.HOME) AND NOT _conn.Referenced THEN
        _M_FaultN(Code := PL_ModuleReasons.ROBOT_NOT_REFERENCED, Text := 'std.error.robotNotReferenced');
        RETURN;
    END_IF
END_IF

CASE _step OF
    10:
        IF _M_IsMotion(Command) THEN
            // MIN(mode ceiling, recipe scale): reduced speed outside automatic is a
            // property of this type, not per-project habit (I.4a(b)).
            _scale := MIN(ParCfg.SpeedCeiling[_conn.ActualMode], ParCmd.SpeedScale);
            _conn.SetSpeedScale(_scale);
        END_IF
        IF NOT _M_Issue() THEN
            // A connector refusal carries its reason in LastResult (link, busy,
            // send) - adopt it VERBATIM (S8.2), never re-classified here. An
            // unchanged reason means nothing was sent at all, which is an
            // unsupported command; adopting the empty diagnostic would erase the
            // fault with a zero code.
            _cd := _conn.LastResult;
            IF _cd.ReasonCode <> _startResult.ReasonCode THEN
                _M_FaultDiag(Diag := _cd);
            ELSE
                _M_Fault(E_Reason.UNSUPPORTED_COMMAND, 'std.error.unsupportedRobotCommand');
            END_IF
            RETURN;
        END_IF
        _tMove(IN := TRUE, PT := SEL(Command = E_RobotCommand.HOME, ParCfg.MoveTimeout, ParCfg.HomeTimeout));
        _step := 20;

    20:
        // (a) the robot own protective stop: abort with ITS OWN reason, kept
        //     deliberately distinct from any S9 safety reason (I.4a(c)).
        IF _conn.ProtectiveStop THEN
            _M_FaultStopped(Code := PL_ModuleReasons.ROBOT_PROTECTIVE_STOP,
                            Text := 'std.error.robotProtectiveStop');
            RETURN;
        END_IF

        // (b) lost permissive -> HELD on-path (I.4b, Core S6.1). Interrupt is sent
        //     ONCE at hold onset; the base re-asserts the hold every scan the
        //     condition is unsatisfied and clears it the scan it returns.
        Intlk();
        IF NOT Intlk.AllOk THEN
            IF NOT _heldOnPath THEN
                _conn.Interrupt();
                _heldOnPath := TRUE;
            END_IF
            _M_HoldDiag(Diag := Intlk.Diagnostic);
            RETURN;
        END_IF
        IF _heldOnPath THEN
            _heldOnPath := FALSE;
            IF _conn.Resumable THEN
                _conn.Resume();
            ELSE
                // The arm left the retained path while held - typically jogged,
                // which is what the pause was for. Resuming would drive through
                // untaught space; refuse loudly instead (I.4b).
                _M_FaultN(Code := PL_ModuleReasons.ROBOT_RESUME_INVALID,
                          Text := 'std.error.robotResumeInvalid');
                RETURN;
            END_IF
        END_IF

        // (c) the connector faulted since the command started: adopt verbatim.
        _cd := _conn.LastResult;
        IF _cd.ReasonCode <> _startResult.ReasonCode THEN
            _M_FaultDiag(Diag := _cd);
            RETURN;
        END_IF

        // (d) completion: accepted, and the arm has stopped moving.
        IF NOT _conn.MotionBusy THEN
            _tMove(IN := FALSE);
            OutCmd.ReachedId := ParCmd.TargetId;
            _M_Complete();
            RETURN;
        END_IF
        IF _tMove.Q THEN
            _M_FaultStopped(Code := PL_ModuleReasons.ROBOT_MOVE_TIMEOUT,
                            Text := 'std.error.robotMoveTimeout');
        END_IF
ELSE
    _M_Fault(E_Reason.STEP_STALLED, 'std.error.undefinedStep');
END_CASE
END_METHOD

// Stop the arm, THEN fault. _M_FaultN raises the reason without touching motion,
// so faulting first would leave a moving robot commanded - the same defect
// FB_AxisCM._M_FaultStopped exists to prevent, and no less serious here.
METHOD PRIVATE _M_FaultStopped
VAR_INPUT
    Code : DINT;
    Text : STRING(255);
END_VAR
IF _conn <> 0 THEN
    _conn.Abort();
END_IF
_M_FaultN(Code := Code, Text := Text);
END_METHOD

// Core S7.2.1 - the application names its own conditions on this module; the
// library declares none. For a robot that matters more than usual: the guard,
// the safe-zone acknowledgement and the "cell clear" are all facts only the
// station can see. Declared conditions start FALSE - declaring one states an
// intent to gate, so a half-wired station holds rather than moves.
METHOD DeclareCondition : BOOL
VAR_INPUT
    Index : INT;
    DescriptionKey : STRING(255);
    Reason : E_Reason;
    Bypassable : BOOL;
END_VAR
IF (Index < 1) OR (Index > PL_Fraktal.MAX_PERMINTLK_COND) THEN
    DeclareCondition := FALSE;
    RETURN;
END_IF
_appCond[Index] := FALSE;
DeclareCondition := Intlk.Define(Index := Index, Description := DescriptionKey,
    Reason := Reason, Bypassable := Bypassable);
END_METHOD

// Drive a condition declared by DeclareCondition, every scan.
METHOD SetCondition : BOOL
VAR_INPUT
    Index : INT;
    Ok : BOOL;
END_VAR
IF (Index < 1) OR (Index > PL_Fraktal.MAX_PERMINTLK_COND) THEN
    SetCondition := FALSE;
    RETURN;
END_IF
_appCond[Index] := Ok;
SetCondition := TRUE;
END_METHOD

METHOD PRIVATE _M_ApplyConditions
VAR
    i : INT;
END_VAR
FOR i := 1 TO PL_Fraktal.MAX_PERMINTLK_COND DO
    Intlk.Cond[i] := _appCond[i];
END_FOR
END_METHOD

// S8.11.4(a) - name the command being timed, so the record reads as an operation
// rather than an enum ordinal. Labels are catalogue keys, resolved by the HMI.
METHOD PRIVATE _M_Tag
CASE Command OF
    E_RobotCommand.POWER_ON:       _M_TagCommand(1,  'std.command.powerOn');
    E_RobotCommand.POWER_OFF:      _M_TagCommand(2,  'std.command.powerOff');
    E_RobotCommand.HOME:           _M_TagCommand(3,  'std.command.home');
    E_RobotCommand.MOVE_TO:        _M_TagCommand(4,  'std.command.moveTo');
    E_RobotCommand.RUN_PATH:       _M_TagCommand(5,  'std.command.robotRunPath');
    E_RobotCommand.RUN_PALLET:     _M_TagCommand(6,  'std.command.robotRunPallet');
    E_RobotCommand.MOVE_TEMPLATE:  _M_TagCommand(7,  'std.command.robotMoveTemplate');
    E_RobotCommand.MOVE_FROM_AREA: _M_TagCommand(8,  'std.command.robotMoveFromArea');
    E_RobotCommand.SET_TOOL:       _M_TagCommand(9,  'std.command.robotSetTool');
    E_RobotCommand.SET_FRAME:      _M_TagCommand(10, 'std.command.robotSetFrame');
    E_RobotCommand.RECONNECT:      _M_TagCommand(11, 'std.command.robotReconnect');
ELSE
    _M_TagCommand(0, '');
END_CASE
END_METHOD

// One ID-addressed primitive per command. FALSE = the connector refused.
METHOD PRIVATE _M_Issue : BOOL
CASE Command OF
    E_RobotCommand.POWER_ON:       _M_Issue := _conn.PowerOn();
    E_RobotCommand.POWER_OFF:      _M_Issue := _conn.PowerOff();
    E_RobotCommand.HOME:           _M_Issue := _conn.Home();
    E_RobotCommand.MOVE_TO:        _M_Issue := _conn.MoveToPoint(ParCmd.TargetId);
    E_RobotCommand.RUN_PATH:       _M_Issue := _conn.RunPath(ParCmd.TargetId, ParCmd.StartIdx, ParCmd.EndIdx);
    E_RobotCommand.RUN_PALLET:     _M_Issue := _conn.RunPallet(ParCmd.TargetId, ParCmd.Nest);
    E_RobotCommand.MOVE_TEMPLATE:  _M_Issue := _conn.MoveTemplate(ParCmd.FromId, ParCmd.TargetId);
    E_RobotCommand.MOVE_FROM_AREA: _M_Issue := _conn.MoveFromArea(ParCmd.TargetId);
    E_RobotCommand.SET_TOOL:       _M_Issue := _conn.SetTool(ParCmd.TargetId);
    E_RobotCommand.SET_FRAME:      _M_Issue := _conn.SetFrame(ParCmd.TargetId);
ELSE
    _M_Issue := FALSE;    // nothing was sent; the dispatch faults unsupported
END_CASE
END_METHOD

// Commands the controller's mode and reference state must permit. POWER_* and
// SET_* are selection, not motion; HOME is sequenced motion and is included.
METHOD PRIVATE _M_IsMotion : BOOL
VAR_INPUT
    Cmd : E_RobotCommand;
END_VAR
_M_IsMotion := (Cmd = E_RobotCommand.HOME)
            OR (Cmd = E_RobotCommand.MOVE_TO)
            OR (Cmd = E_RobotCommand.RUN_PATH)
            OR (Cmd = E_RobotCommand.RUN_PALLET)
            OR (Cmd = E_RobotCommand.MOVE_TEMPLATE)
            OR (Cmd = E_RobotCommand.MOVE_FROM_AREA);
END_METHOD

END_FUNCTION_BLOCK

// ---- FB_SimRobotConnector.TcPOU
// Annex I I.5c - the SIMULATION connector. O6 requires every module to run
// unchanged against simulated or real I/O; for a robot the seam is the connector,
// not the HAL, so without this type a robot CM cannot be virtually commissioned
// at all and a station containing one cannot be dry-run before the arm arrives.
//
// It is deliberately NOT a kinematic simulator and does not pretend to be one.
// What it is faithful about is the CONTRACT: the handshake and its timing, the
// facts it publishes about itself, and its refusals. The pose it reports is a
// plausible synthetic interpolation so displays and area checks have something
// real to move on - never a claim about where an actual arm would be.
//
// Selected as configuration (S2.6): the CM holds I_RobotConnector, so swapping
// this for FB_StaubliVal3Connector changes a declaration and nothing else. That
// is the whole point - simulation is paid once in the connector family, never
// per station (S1.1 O1).
FUNCTION_BLOCK FB_SimRobotConnector EXTENDS FB_DeviceConnectorBase IMPLEMENTS I_RobotConnector
VAR_INPUT
    MoveTime : TIME  := T#200MS;              // how long an accepted motion takes
    HomeTime : TIME  := T#500MS;
    HomeArea : DWORD := 1;                    // area reported once homed (I.11)
    Inject   : E_RobotSimFault;               // I.5c - level, cleared by the caller
END_VAR
VAR
    _busy       : BOOL;
    _referenced : BOOL;
    _powered    : BOOL;
    _protStop   : BOOL;
    _held       : BOOL;
    _mode       : E_RobotOpMode := E_RobotOpMode.AUTO_REMOTE;
    _area       : DWORD;
    _pose       : ST_RobotPose;               // published live pose
    _from       : ST_RobotPose;               // motion start, for interpolation
    _to         : ST_RobotPose;               // motion target
    _tMove      : TON;
    _pt         : TIME;
    _toArea     : DWORD;                      // area that resolves on completion
    _homing     : BOOL;
    _speed      : REAL := 100.0;
    _tool       : DWORD;
    _frame      : DWORD;
    _payload    : DWORD;
    _res        : ST_Diagnostic;              // LastResult
    _ctrl       : ST_Diagnostic;              // ControllerMessage
    _f          : LREAL;
END_VAR

Cyclic();

// No socket to open. The session is up the moment it is asked for, which is
// what makes a dry run start instantly instead of waiting out a backoff.
METHOD PROTECTED _M_Open : BOOL
_M_Open := TRUE;
END_METHOD

METHOD PROTECTED _M_Close : BOOL
_busy := FALSE;
_tMove(IN := FALSE);
_M_Close := TRUE;
END_METHOD

METHOD PROTECTED _M_HbStart : BOOL
_M_HbStart := TRUE;
END_METHOD

// The one place link loss is injected: failing the heartbeat drives the REAL
// loss path in the base - loss confirm, then bounded backoff reconnect - rather
// than a shortcut that would prove nothing about how the cell behaves (I.5c).
METHOD PROTECTED _M_HbPoll : E_HbResult
IF Inject = E_RobotSimFault.LINK_LOSS THEN
    _M_HbPoll := E_HbResult.FAIL;
ELSE
    _M_HbPoll := E_HbResult.OK;
END_IF
END_METHOD

// Advance simulated motion. Override contract: SUPER^ FIRST, so the session,
// heartbeat and reconnect all behave exactly as they do on a real transport.
METHOD Cyclic : BOOL
Cyclic := SUPER^.Cyclic();

// A protective stop is injectable at rest as well as in motion: a crash device
// can trip while the arm is parked, and a cell that only handles the moving case
// discovers that the hard way.
IF Inject = E_RobotSimFault.PROTECTIVE_STOP THEN
    _protStop := TRUE;
    IF _busy THEN
        _busy := FALSE;
        _tMove(IN := FALSE);
    END_IF
END_IF

IF NOT Linked THEN
    // The arm is not commanded from here while the link is down; motion stops
    // rather than silently completing behind a dropped connection.
    _busy := FALSE;
    _tMove(IN := FALSE);
    RETURN;
END_IF

IF _busy AND NOT _held THEN
    _tMove(IN := TRUE, PT := _pt);
    // Plausible pose: linear interpolation start -> target over the move time.
    // Enough for a display to move and for an area check to resolve; never a
    // claim about the path a real arm would take.
    IF _pt > T#0S THEN
        _f := TIME_TO_LREAL(_tMove.ET) / TIME_TO_LREAL(_pt);
    ELSE
        _f := 1.0;
    END_IF
    IF _f > 1.0 THEN
        _f := 1.0;
    END_IF
    _pose.X  := _from.X  + (_to.X  - _from.X)  * _f;
    _pose.Y  := _from.Y  + (_to.Y  - _from.Y)  * _f;
    _pose.Z  := _from.Z  + (_to.Z  - _from.Z)  * _f;
    _pose.RX := _from.RX + (_to.RX - _from.RX) * _f;
    _pose.RY := _from.RY + (_to.RY - _from.RY) * _f;
    _pose.RZ := _from.RZ + (_to.RZ - _from.RZ) * _f;
    IF _tMove.Q THEN
        _tMove(IN := FALSE);
        _busy  := FALSE;
        _pose  := _to;
        _area  := _toArea;
        IF _homing THEN
            _homing     := FALSE;
            _referenced := TRUE;     // homing is what ESTABLISHES the reference
        END_IF
    END_IF
END_IF
END_METHOD

// Refuse with a reason. Every FALSE this type returns leaves a reason behind:
// the CM adopts LastResult verbatim (S8.2), so a silent refusal would surface as
// a fault with a zero code and send the technician nowhere.
METHOD PRIVATE _M_Refuse : BOOL
VAR_INPUT
    Code : DINT;
    Text : STRING(255);
END_VAR
_res.ReasonCode  := Code;
_res.Description := Text;
_res.SourcePath  := Name;
_M_Refuse := FALSE;
END_METHOD

METHOD PRIVATE _M_Accept : BOOL
_res.ReasonCode  := E_Reason.NONE;
_res.Description := '';
_M_Accept := TRUE;
END_METHOD

// Shared gate for everything that reaches the "controller": the link must be up
// and the crash device must not be tripped. Refusals, never queueing (Annex D).
METHOD PRIVATE _M_CanCommand : BOOL
IF NOT Linked THEN
    _M_CanCommand := _M_Refuse(E_Reason.LINK_TIMEOUT, 'std.error.robotLinkDown');
    RETURN;
END_IF
IF _protStop THEN
    _M_CanCommand := _M_Refuse(PL_ModuleReasons.ROBOT_PROTECTIVE_STOP, 'std.error.robotProtectiveStop');
    RETURN;
END_IF
IF _busy THEN
    _M_CanCommand := _M_Refuse(E_Reason.DEVICE_NOT_READY, 'std.error.robotBusy');
    RETURN;
END_IF
_M_CanCommand := TRUE;
END_METHOD

// A deterministic synthetic pose per position ID, so the same ID always reports
// the same place and a test can assert movement without a taught database.
METHOD PRIVATE _M_PoseOf : ST_RobotPose
VAR_INPUT
    PosId : DWORD;
END_VAR
_M_PoseOf.X  := DWORD_TO_LREAL(PosId) * 100.0;
_M_PoseOf.Y  := DWORD_TO_LREAL(PosId) * 50.0;
_M_PoseOf.Z  := 200.0;
_M_PoseOf.RX := 0.0;
_M_PoseOf.RY := 0.0;
_M_PoseOf.RZ := 0.0;
END_METHOD

// Begin a simulated motion toward a position ID. Injected motion failures are
// applied HERE - before anything starts - because I.2's rejection reasons are
// rejections (S5.6), not mid-move surprises.
METHOD PRIVATE _M_Start : BOOL
VAR_INPUT
    ToPosId : DWORD;
    PT      : TIME;
    Routed  : BOOL;     // a template move, which is what NO_ROUTE applies to
END_VAR
IF NOT _M_CanCommand() THEN
    _M_Start := FALSE;
    RETURN;
END_IF
IF NOT _powered THEN
    _M_Start := _M_Refuse(PL_ModuleReasons.ROBOT_CONTROLLER_FAULT, 'std.error.robotNotPowered');
    RETURN;
END_IF
IF Inject = E_RobotSimFault.POINT_UNREACHABLE THEN
    _M_Start := _M_Refuse(PL_ModuleReasons.ROBOT_POINT_UNREACHABLE, 'std.error.robotPointUnreachable');
    RETURN;
END_IF
IF Routed AND (Inject = E_RobotSimFault.NO_ROUTE) THEN
    _M_Start := _M_Refuse(PL_ModuleReasons.ROBOT_NO_ROUTE, 'std.error.robotNoRoute');
    RETURN;
END_IF
_from   := _pose;
_to     := _M_PoseOf(ToPosId);
_toArea := ToPosId;                  // the sim treats each position as its own area
_pt     := PT;
_held   := FALSE;
_busy   := TRUE;
_tMove(IN := FALSE);
_M_Start := _M_Accept();
END_METHOD

METHOD PowerOn : BOOL
IF NOT _M_CanCommand() THEN
    PowerOn := FALSE;
    RETURN;
END_IF
_powered := TRUE;
PowerOn := _M_Accept();
END_METHOD

METHOD PowerOff : BOOL
IF NOT Linked THEN
    PowerOff := _M_Refuse(E_Reason.LINK_TIMEOUT, 'std.error.robotLinkDown');
    RETURN;
END_IF
_powered := FALSE;
_busy    := FALSE;
_tMove(IN := FALSE);
PowerOff := _M_Accept();
END_METHOD

// Homing is what establishes the reference, so it is the one motion that does
// NOT require one - see FB_RobotCM's validation ladder for the matching exemption.
METHOD Home : BOOL
IF NOT _M_Start(ToPosId := 0, PT := HomeTime, Routed := FALSE) THEN
    Home := FALSE;
    RETURN;
END_IF
_homing := TRUE;
_toArea := HomeArea;
Home := TRUE;
END_METHOD

METHOD MoveToPoint : BOOL
VAR_INPUT
    PointId : DWORD;
END_VAR
MoveToPoint := _M_Start(ToPosId := PointId, PT := MoveTime, Routed := FALSE);
END_METHOD

METHOD RunPath : BOOL
VAR_INPUT
    ListId   : DWORD;
    StartIdx : DINT;
    EndIdx   : DINT;
END_VAR
IF EndIdx < StartIdx THEN
    RunPath := _M_Refuse(PL_ModuleReasons.ROBOT_PARAM_OOR, 'std.error.robotPathRangeInvalid');
    RETURN;
END_IF
RunPath := _M_Start(ToPosId := ListId, PT := MoveTime, Routed := FALSE);
END_METHOD

METHOD RunPallet : BOOL
VAR_INPUT
    PalletId : DWORD;
    Nest     : DINT;
END_VAR
IF Nest < 0 THEN
    RunPallet := _M_Refuse(PL_ModuleReasons.ROBOT_PARAM_OOR, 'std.error.robotNestInvalid');
    RETURN;
END_IF
RunPallet := _M_Start(ToPosId := PalletId, PT := MoveTime, Routed := FALSE);
END_METHOD

METHOD MoveTemplate : BOOL
VAR_INPUT
    FromPosId : DWORD;
    ToPosId   : DWORD;
END_VAR
MoveTemplate := _M_Start(ToPosId := ToPosId, PT := MoveTime, Routed := TRUE);
END_METHOD

METHOD MoveFromArea : BOOL
VAR_INPUT
    ToPosId : DWORD;
END_VAR
MoveFromArea := _M_Start(ToPosId := ToPosId, PT := MoveTime, Routed := TRUE);
END_METHOD

// Pause on-path. The retained path is what Resume returns to, and whether it
// is still valid is exactly what NOT_RESUMABLE injects (I.4b).
METHOD Interrupt : BOOL
IF NOT Linked THEN
    Interrupt := _M_Refuse(E_Reason.LINK_TIMEOUT, 'std.error.robotLinkDown');
    RETURN;
END_IF
_held := TRUE;
Interrupt := _M_Accept();
END_METHOD

METHOD Resume : BOOL
IF NOT Linked THEN
    Resume := _M_Refuse(E_Reason.LINK_TIMEOUT, 'std.error.robotLinkDown');
    RETURN;
END_IF
IF NOT Resumable THEN
    Resume := _M_Refuse(PL_ModuleReasons.ROBOT_RESUME_INVALID, 'std.error.robotResumeInvalid');
    RETURN;
END_IF
_held  := FALSE;
Resume := _M_Accept();
END_METHOD

METHOD Abort : BOOL
_busy := FALSE;
_held := FALSE;
_tMove(IN := FALSE);
Abort := _M_Accept();
END_METHOD

// Acknowledge at the "controller" - the crash trip clears here and nowhere else,
// mirroring an arm that will not move again until acknowledged on the pendant.
METHOD ResetController : BOOL
IF NOT Linked THEN
    ResetController := _M_Refuse(E_Reason.LINK_TIMEOUT, 'std.error.robotLinkDown');
    RETURN;
END_IF
_protStop := FALSE;
_ctrl.ReasonCode  := E_Reason.NONE;
_ctrl.Description := '';
ResetController := _M_Accept();
END_METHOD

// The PLC REQUESTS; a real controller grants or does not. The sim grants, but
// never grants UNKNOWN: an uninitialised value must not travel as a request.
METHOD RequestMode : BOOL
VAR_INPUT
    Mode : E_RobotOpMode;
END_VAR
IF Mode = E_RobotOpMode.UNKNOWN THEN
    RequestMode := _M_Refuse(PL_ModuleReasons.ROBOT_MODE_NOT_PERMITTED, 'std.error.robotModeNotPermitted');
    RETURN;
END_IF
IF NOT Linked THEN
    RequestMode := _M_Refuse(E_Reason.LINK_TIMEOUT, 'std.error.robotLinkDown');
    RETURN;
END_IF
_mode := Mode;
RequestMode := _M_Accept();
END_METHOD

METHOD SetSpeedScale : BOOL
VAR_INPUT
    Percent : REAL;
END_VAR
IF (Percent < 0.0) OR (Percent > 100.0) THEN
    SetSpeedScale := _M_Refuse(PL_ModuleReasons.ROBOT_PARAM_OOR, 'std.error.robotSpeedScaleOutOfRange');
    RETURN;
END_IF
_speed := Percent;
SetSpeedScale := _M_Accept();
END_METHOD

METHOD SetTool : BOOL
VAR_INPUT
    ToolId : DWORD;
END_VAR
IF NOT _M_CanCommand() THEN
    SetTool := FALSE;
    RETURN;
END_IF
_tool := ToolId;
SetTool := _M_Accept();
END_METHOD

METHOD SetFrame : BOOL
VAR_INPUT
    FrameId : DWORD;
END_VAR
IF NOT _M_CanCommand() THEN
    SetFrame := FALSE;
    RETURN;
END_IF
_frame := FrameId;
SetFrame := _M_Accept();
END_METHOD

METHOD SetPayload : BOOL
VAR_INPUT
    LoadId : DWORD;
END_VAR
IF NOT _M_CanCommand() THEN
    SetPayload := FALSE;
    RETURN;
END_IF
_payload := LoadId;
SetPayload := _M_Accept();
END_METHOD

// Bounded by the CONTROLLER's reported mode, not by a PLC release alone: jogging
// under automatic is exactly the move nobody is standing ready for.
METHOD Jog : BOOL
VAR_INPUT
    Mode : E_RobotJogMode;
    Axis : INT;
    Dir  : INT;
END_VAR
IF NOT _M_CanCommand() THEN
    Jog := FALSE;
    RETURN;
END_IF
IF (_mode <> E_RobotOpMode.MANUAL_REDUCED) AND (_mode <> E_RobotOpMode.MANUAL_HIGH) THEN
    Jog := _M_Refuse(PL_ModuleReasons.ROBOT_MODE_NOT_PERMITTED, 'std.error.robotModeNotPermitted');
    RETURN;
END_IF
IF (Axis < 1) OR (Dir = 0) THEN
    Jog := _M_Refuse(PL_ModuleReasons.ROBOT_PARAM_OOR, 'std.error.robotJogParamInvalid');
    RETURN;
END_IF
// Jogging leaves the retained path - which is why Resumable goes false.
_pose.X := _pose.X + DINT_TO_LREAL(Dir) * 10.0;
Jog := _M_Accept();
END_METHOD

PROPERTY MotionBusy : BOOL
GET
MotionBusy := _busy;
END_GET
END_PROPERTY

PROPERTY Referenced : BOOL
GET
Referenced := _referenced;
END_GET
END_PROPERTY

// What the controller REPORTS, never what was asked for (I.4a(a)).
PROPERTY ActualMode : E_RobotOpMode
GET
ActualMode := _mode;
END_GET
END_PROPERTY

PROPERTY ActualPosition : ST_RobotPose
GET
ActualPosition := _pose;
END_GET
END_PROPERTY

PROPERTY ControllerMessage : ST_Diagnostic
GET
ControllerMessage := _ctrl;
END_GET
END_PROPERTY

// Resolves through the ordinary area check (I.11): a sim that left this
// unresolved would fail every template move and prove nothing.
PROPERTY CurrentArea : DWORD
GET
CurrentArea := _area;
END_GET
END_PROPERTY

// The robot's OWN crash device - deliberately NOT a S9 safety function.
PROPERTY ProtectiveStop : BOOL
GET
ProtectiveStop := _protStop;
END_GET
END_PROPERTY

// TRUE only while a hold is outstanding and the path is still retained.
PROPERTY Resumable : BOOL
GET
IF Inject = E_RobotSimFault.NOT_RESUMABLE THEN
    Resumable := FALSE;
ELSE
    Resumable := _held AND NOT _protStop;
END_IF
END_GET
END_PROPERTY

PROPERTY LastResult : ST_Diagnostic
GET
LastResult := _res;
END_GET
END_PROPERTY

END_FUNCTION_BLOCK

// ---- FB_AxisCM.TcPOU
// Annex G worked example on the base class: PLCopen Motion behind the standard
// handshake (S10.6). The parent Unit commands MOVE_TO exactly as it commands a
// cylinder EXTEND - it neither knows nor cares that a servo is involved (S6.1).
//
// The drive is reached ONLY through AXIS_REF and Tc2_MC2. That is what makes the
// type drive-agnostic: a Jenny Science XENAX linked as a CiA402 EtherCAT axis, a
// Beckhoff AX5000, or a simulated NC axis are the same code here. Any
// vendor-specific facility belongs in the driver layer (S10.2), never in a
// reusable CM.
//
// Like FB_SeparatorCM this type declares NO interlocks of its own (S7.2.1). Safe
// motion lives in the certified system; this module only READS its status, and
// the application supplies that status - and any station policy - through
// DeclareCondition/SetCondition. A library cannot name "STO cleared" for a
// station it has never seen.
FUNCTION_BLOCK FB_AxisCM EXTENDS FB_ControlModuleBase
VAR_INPUT
    Command : E_AxisCommand;
    ParCfg : ST_AxisParCfg;
    ParCmd : ST_AxisParCmd;
END_VAR
VAR_OUTPUT
    OutCmd : ST_AxisOutCmd;
    OutImm : ST_AxisOutImm;
    Intlk  : FB_PermIntlk;
END_VAR
VAR CONSTANT
    // §3.8b - the layout version of this module's StationCfg. It belongs with
    // the type that owns the structure, not in the reason band. Bump it when a
    // member is added or its meaning changes (§13).
    AXIS_STATIONCFG_SCHEMA : UINT := 2;   // v2 added JogRequiresEnable
END_VAR
VAR PERSISTENT
    // §3.8b - the retained image. PERSISTENT is the BACKING, not the architecture:
    // the value is registered per (Scope, WriteKey) like every other editable
    // value, so when a set store (file/JSON/XML, MES, asset system) is wired it
    // projects this through the same walk with no change here.
    // Only the VALUE is persistent - the registry's pTarget stays in ordinary
    // VAR, because a retained POINTER names nothing after a restart
    // (ST_ConfigWriteDef, TC3 §3.8b).
    _station : ST_AxisStationCfg;
END_VAR
VAR
    {attribute 'OPC.UA.DA' := '0'}
    _axis : REFERENCE TO AXIS_REF;
    {attribute 'OPC.UA.DA' := '0'}
    _recipe : I_RecipeProvider;
    {attribute 'OPC.UA.DA' := '0'}
    _power : MC_Power;
    {attribute 'OPC.UA.DA' := '0'}
    _homeFb : MC_Home;
    {attribute 'OPC.UA.DA' := '0'}
    _moveFb : MC_MoveAbsolute;
    {attribute 'OPC.UA.DA' := '0'}
    _stopFb : MC_Stop;
    {attribute 'OPC.UA.DA' := '0'}
    _resetFb : MC_Reset;
    {attribute 'OPC.UA.DA' := '0'}
    _jogFb : MC_Jog;
    _jogSeen   : BOOL;   // a held request arrived THIS scan (freshness, O10)
    _jogReqDir : INT;    // +1 / -1 / 0 as last asked
    _jogEnabled: BOOL;   // an enabling device was held when it was asked
    _jogDriving: BOOL;   // the axis is being jogged right now
    _tJogStale : TON;
    _tMove : TON;
    _homed : BOOL;
    _parCfgStaged : ST_AxisParCfg;
    _recipePrepared : BOOL;
    _appCond : ARRAY[1..PL_Fraktal.MAX_PERMINTLK_COND] OF BOOL;
END_VAR

Cyclic();

METHOD PROTECTED OnCyclic : DINT
OnCyclic := SUPER^.OnCyclic();
_M_ApplyConditions();
Intlk();
IF __ISVALIDREF(_axis) THEN                  // defensive (S5.6) [TC3]
    // Enable follows the declared conditions. Losing one drops the enable in the
    // same scan it is lost; re-enabling after it returns is a deliberate command,
    // never automatic (S9.3, S9.4).
    _power(Axis := _axis, Enable := Intlk.AllOk, Enable_Positive := Intlk.AllOk,
        Enable_Negative := Intlk.AllOk, Override := 100.0);
    OutImm.ActPos := _axis.NcToPlc.ActPos;
    OutImm.ActVelocity := _axis.NcToPlc.ActVelo;
    OutImm.DriveEnabled := _power.Status;
END_IF
_M_JogCyclic();
OutImm.TaughtPosition := _station.TaughtPosition;
OutImm.Homed := _homed;
OutCmd.Homed := _homed;
END_METHOD

METHOD PRIVATE _M_ApplyConditions
VAR
    i : INT;
END_VAR
FOR i := 1 TO PL_Fraktal.MAX_PERMINTLK_COND DO
    Intlk.Cond[i] := _appCond[i];
END_FOR
END_METHOD

